(* IEC 61131-3 sources: SmartHomeNew/ (part 2) *)

(* ---- GVL_DEBUG_VIEW.gvl ---- *)
VAR_GLOBAL
    D_Current_Time_MS : UDINT := 0;

    D_Safety_Mode : E_Safety_Mode := NORMAL;
    D_Safety_Active : BOOL := FALSE;
    D_Recovery_Phase : E_Recovery_Phase := IDLE;
    D_Recovery_Active : BOOL := FALSE;
    D_Recovery_Exit_Allowed : BOOL := FALSE;
    D_Authority_Revocation_Active : BOOL := FALSE;
    D_Authority_Restoration_Allowed : BOOL := FALSE;
    D_Authority_Restoration_Completed : BOOL := FALSE;

    D_Current_Scenario : STRING(255) := '';
    D_Behavior_Reason : STRING(255) := '';
    D_Score_Night : INT := 0;
    D_Score_Preheat : INT := 0;
    D_Score_VentBoost : INT := 0;
    D_Score_AccessSecure : INT := 0;
    D_Intent_Night : BOOL := FALSE;
    D_Intent_Comfort : BOOL := FALSE;
    D_Intent_VentBoost : BOOL := FALSE;
    D_Intent_AccessSecure : BOOL := FALSE;

    D_Heating_Block : BOOL := FALSE;
    D_Vent_Stop : BOOL := FALSE;
    D_Water_Block : BOOL := FALSE;
    D_Access_Open_Active : BOOL := FALSE;

    D_Global_Reason : STRING(255) := '';
    D_Behavior_Why_Active : STRING(255) := '';
    D_Heating_Why_Blocked : STRING(255) := '';
    D_Vent_Why_Stopped : STRING(255) := '';
    D_Water_Why_Closed : STRING(255) := '';
    D_Access_Why_Opened : STRING(255) := '';

    D_Main_VentBoost_Zone : INT := 0;
    D_Main_VentBoost_Zone_Weight : REAL := 0.0;
    D_Main_VentBoost_Zone_Confidence : REAL := 0.0;
    D_Max_VentBoost_Zone_Weight : REAL := 0.0;
    D_Min_VentBoost_Zone_Weight : REAL := 0.0;

    // MAIN phase feedback summary.
    D_Main_Phase_Current : UINT := 0;
    D_Main_Phase_Critical_Executed : BOOL := FALSE;
    D_Main_Phase_Critical_Valid : BOOL := FALSE;
    D_Main_Phase_Observability_Executed : BOOL := FALSE;
    D_Main_Phase_Observability_Valid : BOOL := FALSE;
    D_Main_Phase_Any_Invalid : BOOL := FALSE;
    D_Main_Phase_Any_Skipped_By_Design : BOOL := FALSE;
    D_Main_Phase_Status_Code : UINT := 0;
    D_Main_Phase_Status_Text : STRING(160) := '';

    // Domain execution policy summary.
    D_Domain_Policy_Any_Critical : BOOL := FALSE;
    D_Domain_Policy_Any_Periodic : BOOL := FALSE;
    D_Domain_Policy_Any_Periodic_Due : BOOL := FALSE;
    D_Domain_Policy_Any_Idle : BOOL := FALSE;
    D_Domain_Policy_Status_Code : UINT := 0;
    D_Domain_Policy_Status_Text : STRING(160) := '';

    D_Access_Mode : UINT := 0;
    D_Access_Critical_Run : BOOL := FALSE;
    D_Access_Periodic_Run : BOOL := FALSE;
    D_Access_Periodic_Due : BOOL := FALSE;
    D_Access_Idle_By_Design : BOOL := FALSE;

    D_Lighting_Mode : UINT := 0;
    D_Lighting_Critical_Run : BOOL := FALSE;
    D_Lighting_Periodic_Run : BOOL := FALSE;
    D_Lighting_Periodic_Due : BOOL := FALSE;
    D_Lighting_Idle_By_Design : BOOL := FALSE;

    D_Water_Mode : UINT := 0;
    D_Water_Critical_Run : BOOL := FALSE;
    D_Water_Periodic_Run : BOOL := FALSE;
    D_Water_Periodic_Due : BOOL := FALSE;
    D_Water_Idle_By_Design : BOOL := FALSE;

    D_Heating_Mode : UINT := 0;
    D_Heating_Critical_Run : BOOL := FALSE;
    D_Heating_Periodic_Run : BOOL := FALSE;
    D_Heating_Periodic_Due : BOOL := FALSE;
    D_Heating_Idle_By_Design : BOOL := FALSE;

    D_Vent_Mode : UINT := 0;
    D_Vent_Critical_Run : BOOL := FALSE;
    D_Vent_Periodic_Run : BOOL := FALSE;
    D_Vent_Periodic_Due : BOOL := FALSE;
    D_Vent_Idle_By_Design : BOOL := FALSE;

    D_Simulation_Mode : UINT := 0;
    D_Simulation_Run_Allowed : BOOL := FALSE;
    D_Simulation_Periodic_Due : BOOL := FALSE;
    D_Simulation_Idle_By_Design : BOOL := FALSE;

    // Domain execution validation summary.
    D_Domain_Validation_Executed : BOOL := FALSE;
    D_Domain_Validation_Valid : BOOL := FALSE;
    D_Domain_Validation_Any_Stale_Output_Risk : BOOL := FALSE;
    D_Domain_Validation_Any_Policy_Mismatch : BOOL := FALSE;
    D_Access_Stale_Output_Risk : BOOL := FALSE;
    D_Lighting_Stale_Output_Risk : BOOL := FALSE;
    D_Water_Stale_Output_Risk : BOOL := FALSE;
    D_Heating_Stale_Output_Risk : BOOL := FALSE;
    D_Vent_Stale_Output_Risk : BOOL := FALSE;
    D_Domain_Validation_Status_Code : UINT := 0;
    D_Domain_Validation_Status_Text : STRING(160) := '';

    // Runtime scenario validation summary.
    D_Runtime_Scenario_Validation_Executed : BOOL := FALSE;
    D_Runtime_Scenario_Validation_Valid : BOOL := FALSE;
    D_Runtime_Scenario_Any_Context_Invalid : BOOL := FALSE;
    D_Runtime_Idle_Context_Active : BOOL := FALSE;
    D_Runtime_Security_Context_Active : BOOL := FALSE;
    D_Runtime_Away_Context_Active : BOOL := FALSE;
    D_Runtime_Presence_Context_Active : BOOL := FALSE;
    D_Runtime_Fire_Context_Active : BOOL := FALSE;
    D_Runtime_Gas_Context_Active : BOOL := FALSE;
    D_Runtime_Leak_Context_Active : BOOL := FALSE;
    D_Runtime_Global_Stop_Context_Active : BOOL := FALSE;
    D_Runtime_Freeze_Context_Active : BOOL := FALSE;
    D_Runtime_Heating_Context_Valid : BOOL := FALSE;
    D_Runtime_Vent_Context_Valid : BOOL := FALSE;
    D_Runtime_Access_Context_Valid : BOOL := FALSE;
    D_Runtime_Global_Stop_Context_Valid : BOOL := FALSE;
    D_Runtime_Scenario_Status_Code : UINT := 0;
    D_Runtime_Scenario_Status_Text : STRING(160) := '';

    // Runtime physical IO validation summary.
    D_Runtime_IO_Validation_Executed : BOOL := FALSE;
    D_Runtime_IO_Validation_Valid : BOOL := FALSE;
    D_Runtime_IO_Any_Invalid : BOOL := FALSE;
    D_Runtime_IO_Fire_Valid : BOOL := FALSE;
    D_Runtime_IO_Gas_Valid : BOOL := FALSE;
    D_Runtime_IO_Leak_Valid : BOOL := FALSE;
    D_Runtime_IO_Global_Stop_Valid : BOOL := FALSE;
    D_Runtime_IO_Inactive_PLC_Valid : BOOL := FALSE;
    D_Runtime_IO_Freeze_Valid : BOOL := FALSE;
    D_Runtime_IO_Status_Code : UINT := 0;
    D_Runtime_IO_Status_Text : STRING(160) := '';

    // HMI / dashboard sensor quality view.
    D_Input_Source_Valid : BOOL := FALSE;
    D_Input_Degraded : BOOL := FALSE;
    D_Sensor_Fault : BOOL := FALSE;
    D_Validation_Failed : BOOL := FALSE;
    D_Anomaly_Detected : BOOL := FALSE;
    D_Validation_Reason : STRING(120) := '';
    D_Anomaly_Reason : STRING(120) := '';
    D_Last_Invalid_Zone : INT := 0;
    D_Min_Zone_Confidence : REAL := 1.0;
    D_Worst_Zone : INT := 0;

    // Runtime diagnostics formerly stored in legacy GVL_TEST.
    D_Ownership_Violation : BOOL := FALSE;

    D_Adapt_Profile : E_Adapt_Profile := ADAPT_PROFILE_BALANCED;
    D_Adapt_Profile_Text : STRING(32) := 'BALANCED';

    D_Last_Trace_Text : STRING(120) := '';
    D_Last_Trace_Time_MS : UDINT := 0;
    D_Last_Trace_Reason : E_System_Reason_Code := REASON_NONE;
END_VAR

(* ---- GVL_DIAGNOSTICS_EXT.gvl ---- *)
{attribute 'qualified_only'}
VAR_GLOBAL
    // Health scores (0..1)
    G_Health_Heating : REAL := 1.0;
    G_Health_Safety : REAL := 1.0;
    G_Health_IO : REAL := 1.0;

    // Error counters
    G_Error_Count_Heating : UDINT := 0;
    G_Error_Count_Safety : UDINT := 0;
    G_Error_Count_IO : UDINT := 0;

    // Last error timestamps
    G_Last_Error_Time_Heating : UDINT := 0;
    G_Last_Error_Time_Safety : UDINT := 0;
    G_Last_Error_Time_IO : UDINT := 0;

    // Timing
    G_Last_Update_Time : UDINT := 0;

    // Cycle / watchdog statistics (interval between diagnostics executions)
    G_Cycle_Expected_MS : UDINT := 250;
    G_Cycle_Warning_MS : UDINT := 375;
    G_Cycle_Critical_MS : UDINT := 500;
    G_Cycle_Last_MS : UDINT := 0;
    G_Cycle_Max_MS : UDINT := 0;
    G_Cycle_Min_MS : UDINT := 0;
    G_Cycle_Avg_MS : REAL := 0.0;
    G_Cycle_Sample_Count : UDINT := 0;
    G_Cycle_Overrun_Count : UDINT := 0;
    G_Cycle_Critical_Count : UDINT := 0;
    G_Cycle_Last_Overrun_MS : UDINT := 0;
    G_Cycle_Last_Overrun_Time_MS : UDINT := 0;
    G_Cycle_Overrun_Active : BOOL := FALSE;
    G_Cycle_Critical_Active : BOOL := FALSE;

    // Compact degraded state mirrors.
    G_Heating_State : INT := 0; // 0=OK,1=DEGRADED,2=CRITICAL
    G_Safety_State : INT := 0;
    G_IO_State : INT := 0;
END_VAR

(* ---- GVL_Distributed_Authority.gvl ---- *)
{attribute 'qualified_only'}
VAR_GLOBAL RETAIN
    G_Authority_State : ST_Distributed_Authority_State;

    G_Master_Controller_Id : UINT;
    G_Backup_Controller_Id : UINT;

    G_Authority_Lease_Start_MS : UDINT;
    G_Authority_Lease_Duration_MS : UDINT := 30000;
END_VAR

VAR_GLOBAL
    G_Runtime_Valid : BOOL;
    G_Last_Update_MS : UDINT;

    G_Split_Brain_Blocked : BOOL;
    G_Distributed_Safety_Barrier_OK : BOOL;

    G_Status_Code : UINT;
    G_Status_Text : STRING(160);
END_VAR

(* ---- GVL_DISTRIBUTED_COMMIT.gvl ---- *)
VAR_GLOBAL
    // ======================================================
    // DISTRIBUTED PUBLICATION COMMIT STATE
    // ======================================================
    // Deterministic peer publication commit handshake foundation.
    // Publication-continuity governance only.
    // Does not invalidate runtime barrier, PLC fencing
    // or local immutable snapshot authority.
    // ======================================================

    Distributed_Commit_Epoch : ULINT := 0;
    Distributed_Commit_Reconciliation_Epoch : ULINT := 0;

    Local_Publication_Commit_Epoch : ULINT := 0;
    Peer_Publication_Commit_Epoch : ULINT := 0;

    Local_Prepare_Epoch : ULINT := 0;
    Peer_Prepare_Epoch : ULINT := 0;

    Local_Commit_Token : ULINT := 0;
    Peer_Commit_Token : ULINT := 0;

    Publication_Prepare_Active : BOOL := FALSE;
    Publication_Prepare_Valid : BOOL := FALSE;
    Publication_Commit_Requested : BOOL := FALSE;
    Publication_Commit_Confirmed : BOOL := FALSE;

    Peer_Commit_Ack_Valid : BOOL := FALSE;
    Peer_Commit_Ack_Expired : BOOL := FALSE;
    Peer_Commit_Mismatch : BOOL := FALSE;
    Peer_Commit_Replay_Detected : BOOL := FALSE;
    Peer_Commit_Missing : BOOL := FALSE;

    Commit_Lease_Active : BOOL := FALSE;
    Commit_Lease_Expired : BOOL := FALSE;
    Commit_Timeout_MS : UDINT := 5000;

    Local_Commit_Last_Refresh_MS : UDINT := 0;
    Peer_Commit_Last_Refresh_MS : UDINT := 0;
    Commit_Last_Reconciliation_MS : UDINT := 0;

    Distributed_Commit_Valid : BOOL := FALSE;
    Distributed_Commit_Quarantine_Active : BOOL := FALSE;

    Distributed_Commit_Last_Error_Code : UDINT := 0;
    Distributed_Commit_Last_Error_Text : STRING(160) := '';
END_VAR

(* ---- GVL_DISTRIBUTED_EPOCH.gvl ---- *)
VAR_GLOBAL
    // ======================================================
    // DISTRIBUTED EPOCH CONSISTENCY STATE
    // ======================================================
    // Centralized peer epoch reconciliation foundation.
    // Prevents distributed stale authority and split-brain continuity.
    // ======================================================

    Distributed_Epoch : ULINT := 0;
    Distributed_Reconciliation_Epoch : ULINT := 0;

    Local_Runtime_Epoch : ULINT := 0;
    Peer_Runtime_Epoch : ULINT := 0;

    Local_Snapshot_Epoch : ULINT := 0;
    Peer_Snapshot_Epoch : ULINT := 0;

    Local_Boot_Generation : ULINT := 0;
    Peer_Boot_Generation : ULINT := 0;

    Local_Fencing_Token : ULINT := 0;
    Peer_Fencing_Token : ULINT := 0;

    Distributed_Epoch_Consistent : BOOL := FALSE;
    Distributed_Reconciliation_Valid : BOOL := FALSE;
    Distributed_Publication_Allowed : BOOL := FALSE;

    Peer_Lease_Active : BOOL := FALSE;
    Peer_Lease_Expired : BOOL := FALSE;
    Peer_Lease_Timeout_MS : UDINT := 5000;

    Peer_Last_Refresh_MS : UDINT := 0;
    Peer_Last_Reconciliation_MS : UDINT := 0;

    Peer_Snapshot_Stale : BOOL := FALSE;
    Peer_Runtime_Stale : BOOL := FALSE;
    Peer_Boot_Mismatch : BOOL := FALSE;
    Peer_Fencing_Conflict : BOOL := FALSE;
    Peer_Semantic_Continuity_Lost : BOOL := FALSE;

    Distributed_Quarantine_Active : BOOL := FALSE;

    Distributed_Last_Error_Code : UDINT := 0;
    Distributed_Last_Error_Text : STRING(160) := '';
END_VAR

(* ---- GVL_Distributed_Orchestration.gvl ---- *)
{attribute 'qualified_only'}
VAR_GLOBAL
    G_Topology_Domain : ARRAY[1..32] OF ST_Distributed_Topology_Domain;
    G_Orchestration_State : ST_Distributed_Orchestration_State;
END_VAR

VAR_GLOBAL RETAIN
    G_Last_Distributed_Sequence_Id : UDINT;
END_VAR

VAR_GLOBAL
    G_Runtime_Valid : BOOL;
    G_Last_Update_MS : UDINT;

    G_Cross_Node_Isolation_Active : BOOL;
    G_Cross_Node_Recovery_Active : BOOL;
    G_Cross_Node_Rollback_Active : BOOL;

    G_Distributed_Projection_Healthy : BOOL;
    G_Distributed_Scheduler_Healthy : BOOL;

    G_Status_Code : UINT;
    G_Status_Text : STRING(160);
END_VAR

(* ---- GVL_Distributed_Projection_Ownership.gvl ---- *)
{attribute 'qualified_only'}
VAR_GLOBAL RETAIN
    G_Projection_Ownership : ARRAY[1..128] OF ST_Distributed_Projection_Ownership;
END_VAR

VAR_GLOBAL
    G_Runtime_Valid : BOOL;
    G_Last_Update_MS : UDINT;

    G_Any_Ownership_Conflict : BOOL;
    G_Any_Ownership_Stale : BOOL;
    G_Any_Projection_Blocked : BOOL;

    G_Status_Code : UINT;
    G_Status_Text : STRING(160);
END_VAR

(* ---- GVL_Distributed_Runtime.gvl ---- *)
{attribute 'qualified_only'}
VAR_GLOBAL RETAIN
    // Keep only compact continuity metadata in non-volatile memory.
    // Runtime node/session/message state is rebuilt by the distributed
    // supervisor chain during cyclic execution and must not consume RETAIN.
    G_Last_Replication_Sequence_Id : UDINT;
END_VAR

VAR_GLOBAL
    G_Local_Node_State : ST_Distributed_Runtime_Node_State;
    G_Remote_Node_State : ARRAY[1..8] OF ST_Distributed_Runtime_Node_State;

    G_Replication_TX : ARRAY[1..64] OF ST_Distributed_Runtime_Message;
    G_Replication_RX : ARRAY[1..64] OF ST_Distributed_Runtime_Message;

    G_Runtime_Valid : BOOL;
    G_Last_Update_MS : UDINT;

    G_Any_Remote_Node_Degraded : BOOL;
    G_Any_Remote_Node_Offline : BOOL;
    G_Split_Brain_Suspected : BOOL;

    G_Distributed_Authority_Healthy : BOOL;
    G_Distributed_Replication_Healthy : BOOL;

    G_Status_Code : UINT;
    G_Status_Text : STRING(160);
END_VAR

(* ---- GVL_DISTRIBUTED_SNAPSHOT.gvl ---- *)
VAR_GLOBAL
    // ======================================================
    // DISTRIBUTED IMMUTABLE SNAPSHOT STATE
    // ======================================================
    // Peer immutable publication snapshot reconciliation.
    // Publication-authoritative only: does not invalidate
    // runtime barrier, PLC fencing or local snapshot freeze.
    // ======================================================

    Distributed_Snapshot_Epoch : ULINT := 0;
    Distributed_Snapshot_Reconciliation_Epoch : ULINT := 0;

    Local_Distributed_Snapshot_Epoch : ULINT := 0;
    Peer_Distributed_Snapshot_Epoch : ULINT := 0;

    Local_Runtime_Snapshot_Epoch : ULINT := 0;
    Peer_Runtime_Snapshot_Epoch : ULINT := 0;

    Local_Publication_Epoch : ULINT := 0;
    Peer_Publication_Epoch : ULINT := 0;

    Distributed_Snapshot_Frozen : BOOL := FALSE;
    Peer_Snapshot_Immutable : BOOL := FALSE;

    Distributed_Publication_Reconciled : BOOL := FALSE;
    Distributed_Publication_Freeze_Valid : BOOL := FALSE;
    Distributed_Snapshot_Consistent : BOOL := FALSE;

    Peer_Publication_Stale : BOOL := FALSE;
    Peer_Snapshot_Not_Immutable : BOOL := FALSE;
    Peer_Publication_Divergence : BOOL := FALSE;
    Peer_Publication_Reconciliation_Lost : BOOL := FALSE;

    Distributed_Snapshot_Quarantine_Active : BOOL := FALSE;

    Peer_Snapshot_Last_Refresh_MS : UDINT := 0;
    Peer_Snapshot_Lease_Active : BOOL := FALSE;
    Peer_Snapshot_Lease_Expired : BOOL := FALSE;
    Peer_Snapshot_Lease_Timeout_MS : UDINT := 5000;

    Distributed_Snapshot_Last_Error_Code : UDINT := 0;
    Distributed_Snapshot_Last_Error_Text : STRING(160) := '';
END_VAR

(* ---- GVL_DOMAIN_EXECUTION_POLICY.gvl ---- *)
{attribute 'qualified_only'}
VAR_GLOBAL
    // Domain execution policy. Observational first layer.
    // This GVL classifies when a domain needs critical, periodic or idle execution.
    // It does not directly control physical outputs.

    G_Last_Update_MS : UDINT := 0;

    // Scenario/context classification.
    G_Security_Context_Active : BOOL := FALSE;
    G_Away_Context_Active : BOOL := FALSE;
    G_Presence_Context_Active : BOOL := FALSE;
    G_Emergency_Context_Active : BOOL := FALSE;

    // Periodic observation intervals.
    Access_Periodic_Interval_MS : UDINT := 1000;
    Lighting_Periodic_Interval_MS : UDINT := 1000;
    Water_Periodic_Interval_MS : UDINT := 1000;
    Heating_Periodic_Interval_MS : UDINT := 5000;
    Vent_Periodic_Interval_MS : UDINT := 3000;
    Simulation_Periodic_Interval_MS : UDINT := 1000;

    // Access.
    Access_Critical_Run : BOOL := FALSE;
    Access_Periodic_Run : BOOL := FALSE;
    Access_Periodic_Due : BOOL := FALSE;
    Access_Idle_By_Design : BOOL := FALSE;

    // Lighting.
    Lighting_Critical_Run : BOOL := FALSE;
    Lighting_Periodic_Run : BOOL := FALSE;
    Lighting_Periodic_Due : BOOL := FALSE;
    Lighting_Idle_By_Design : BOOL := FALSE;

    // Water.
    Water_Critical_Run : BOOL := FALSE;
    Water_Periodic_Run : BOOL := FALSE;
    Water_Periodic_Due : BOOL := FALSE;
    Water_Idle_By_Design : BOOL := FALSE;

    // Heating.
    Heating_Critical_Run : BOOL := FALSE;
    Heating_Periodic_Run : BOOL := FALSE;
    Heating_Periodic_Due : BOOL := FALSE;
    Heating_Idle_By_Design : BOOL := FALSE;

    // Ventilation.
    Vent_Critical_Run : BOOL := FALSE;
    Vent_Periodic_Run : BOOL := FALSE;
    Vent_Periodic_Due : BOOL := FALSE;
    Vent_Idle_By_Design : BOOL := FALSE;

    // Simulation.
    Simulation_Context_Active : BOOL := FALSE;
    Simulation_Run_Allowed : BOOL := FALSE;
    Simulation_Periodic_Due : BOOL := FALSE;
    Simulation_Idle_By_Design : BOOL := FALSE;

    // Summary.
    Any_Critical_Run : BOOL := FALSE;
    Any_Periodic_Run : BOOL := FALSE;
    Any_Periodic_Due : BOOL := FALSE;
    Any_Idle_By_Design : BOOL := FALSE;
    Status_Code : UINT := 0;
    Status_Text : STRING(160) := '';
END_VAR

(* ---- GVL_DOMAIN_EXECUTION_VALIDATION.gvl ---- *)
{attribute 'qualified_only'}
VAR_GLOBAL
    // Domain execution validation. Observational only.
    // Detects policy/output mismatches before runtime gating is trusted.

    G_Last_Update_MS : UDINT := 0;
    G_Validation_Executed : BOOL := FALSE;
    G_Validation_Valid : BOOL := TRUE;

    Access_Stale_Output_Risk : BOOL := FALSE;
    Lighting_Stale_Output_Risk : BOOL := FALSE;
    Water_Stale_Output_Risk : BOOL := FALSE;
    Heating_Stale_Output_Risk : BOOL := FALSE;
    Vent_Stale_Output_Risk : BOOL := FALSE;

    Any_Stale_Output_Risk : BOOL := FALSE;
    Any_Policy_Mismatch : BOOL := FALSE;
    Status_Code : UINT := 0;
    Status_Text : STRING(160) := '';
END_VAR

(* ---- GVL_ENERGY_ISOLATION_CAUSALITY_FABRIC.gvl ---- *)
VAR_GLOBAL
    Energy_Isolation_Causality_Valid : BOOL := FALSE;
    Energy_Isolation_Causality_Granted : BOOL := FALSE;

    Physical_Energy_Isolation_Valid : BOOL := FALSE;
    Unsafe_Energy_Propagation_Prevented : BOOL := FALSE;
    CrossDomain_Power_Segmentation_Canonical : BOOL := FALSE;
    Energy_Isolation_Lineage_Coherent : BOOL := FALSE;

    Energy_Causality_Grounded : BOOL := FALSE;
    Distributed_Energy_Isolation_Consensus : BOOL := FALSE;

    Residual_Energy_Leakage_Detected : BOOL := FALSE;
    CrossDomain_Power_Backfeed_Detected : BOOL := FALSE;
    SplitEnergy_Topology_Detected : BOOL := FALSE;
    Unsafe_Energy_Propagation_Detected : BOOL := FALSE;

    Energy_Isolation_Epoch : UDINT := 0;
END_VAR

(* ---- GVL_EPISTEMIC_INTEGRITY_FABRIC.gvl ---- *)
VAR_GLOBAL
    // Global deterministic epistemic integrity authority.
    Epistemic_Integrity_Valid : BOOL := FALSE;
    Epistemic_Integrity_Granted : BOOL := FALSE;
    Epistemic_Integrity_Quarantine_Active : BOOL := TRUE;

    // Physical reality anchoring proofs.
    Physical_Reality_Model_Coherent : BOOL := FALSE;
    Sensor_Truth_Consensus_Valid : BOOL := FALSE;
    Telemetry_Reality_Alignment_Stable : BOOL := FALSE;
    Distributed_Reality_Model_Consistent : BOOL := FALSE;
    Causal_Model_Physically_Valid : BOOL := FALSE;

    // Long-term epistemic integrity.
    Historical_Reality_Anchoring_Valid : BOOL := FALSE;
    Physical_Truth_Lineage_Coherent : BOOL := FALSE;
    Reality_Model_Drift_Bounded : BOOL := FALSE;
    Semantic_To_Physical_Causality_Valid : BOOL := FALSE;

    // Epistemic split-brain detectors.
    Physically_False_Consensus_Detected : BOOL := FALSE;
    Telemetry_Corruption_Coherent_Detected : BOOL := FALSE;
    Historical_Reality_Divergence_Detected : BOOL := FALSE;
    Sensor_Trust_Erosion_Detected : BOOL := FALSE;
    Causal_Model_Poisoning_Detected : BOOL := FALSE;
    LongTerm_Epistemic_Drift_Detected : BOOL := FALSE;

    // Epistemic epochs.
    Epistemic_Integrity_Epoch : UDINT := 0;
    Epistemic_Integrity_Epoch_Coherent : BOOL := FALSE;

    // Temporal authority.
    Epistemic_Integrity_Last_Update_MS : UDINT := 0;
    Epistemic_Integrity_Lease_Expired : BOOL := TRUE;

    // Diagnostics.
    Epistemic_Integrity_Last_Error_Code : UDINT := 0;
    Epistemic_Integrity_Last_Error_Text : STRING(160) := '';
    Epistemic_Integrity_Invalidation_Count : UDINT := 0;
END_VAR

(* ---- GVL_EXECUTION_PROGRESS_CAUSALITY_FABRIC.gvl ---- *)
VAR_GLOBAL
    Execution_Progress_Causality_Valid : BOOL := FALSE;
    Execution_Progress_Causality_Granted : BOOL := FALSE;

    Progress_Causality_Grounded : BOOL := FALSE;
    Deterministic_Execution_Continuation_Valid : BOOL := FALSE;
    Progress_Lineage_Coherent : BOOL := FALSE;

    Distributed_Progress_Convergence_Valid : BOOL := FALSE;
    Progress_Timeline_Monotonic : BOOL := FALSE;

    Distributed_Execution_Stall_Detected : BOOL := FALSE;
    Execution_Progress_Divergence_Detected : BOOL := FALSE;
    Recovery_Progress_Oscillation_Detected : BOOL := FALSE;

    Execution_Progress_Epoch : UDINT := 0;
END_VAR

(* ---- GVL_EXECUTION_PROJECTION_INTEGRITY_FABRIC.gvl ---- *)
VAR_GLOBAL
    // Deterministic execution projection integrity governance.
    Execution_Projection_Integrity_Valid : BOOL := FALSE;
    Execution_Projection_Integrity_Granted : BOOL := FALSE;
    Execution_Projection_Integrity_Quarantine_Active : BOOL := TRUE;

    // Governance-to-execution projection proofs.
    Execution_Authority_Projection_Consistent : BOOL := FALSE;
    CrossDomain_Actuation_Enforcement_Aligned : BOOL := FALSE;
    Physical_Execution_Governance_Canonical : BOOL := FALSE;
    Actuation_Surface_Consensus_Valid : BOOL := FALSE;
    Execution_Projection_Lineage_Coherent : BOOL := FALSE;

    // Execution enforcement integrity.
    Runtime_Actuation_Projection_Stable : BOOL := FALSE;
    Distributed_Execution_Equivalence_Valid : BOOL := FALSE;
    Execution_Governance_Causality_Grounded : BOOL := FALSE;
    Physical_Enforcement_Timeline_Monotonic : BOOL := FALSE;

    // Execution projection split-brain detectors.
    Execution_Projection_Divergence_Detected : BOOL := FALSE;
    Actuation_Path_Authority_Bypass_Detected : BOOL := FALSE;
    CrossDomain_Enforcement_Fork_Detected : BOOL := FALSE;
    Canonical_Governance_Execution_Lost : BOOL := FALSE;
    Runtime_Execution_Lineage_Drift_Detected : BOOL := FALSE;
    Distributed_Actuation_Reality_Fork_Detected : BOOL := FALSE;

    // Execution epochs.
    Execution_Projection_Integrity_Epoch : UDINT := 0;
    Execution_Projection_Integrity_Epoch_Coherent : BOOL := FALSE;

    // Temporal authority.
    Execution_Projection_Integrity_Last_Update_MS : UDINT := 0;
    Execution_Projection_Integrity_Lease_Expired : BOOL := TRUE;

    // Diagnostics.
    Execution_Projection_Integrity_Last_Error_Code : UDINT := 0;
    Execution_Projection_Integrity_Last_Error_Text : STRING(160) := '';
    Execution_Projection_Integrity_Invalidation_Count : UDINT := 0;
END_VAR

(* ---- GVL_External_Monitoring.gvl ---- *)
VAR_GLOBAL
    // === EXTERNAL SHADOW POLICY CONTRACT ===
    G_Shadow_Any_Alert_Active : BOOL;
    G_Shadow_CO_Active : BOOL;
    G_Shadow_Methane_Active : BOOL;
    G_Shadow_Smoke_Active : BOOL;

    G_Shadow_CO_Healthy : BOOL;
    G_Shadow_Methane_Healthy : BOOL;
    G_Shadow_Smoke_Healthy : BOOL;

    G_Shadow_Dominant_Channel : STRING(32);
    G_Shadow_Policy_Summary_Text : STRING(160);
    G_Shadow_Recent_Activity_Text : STRING(160);
    G_Shadow_Rate_Summary_Text : STRING(160);
    G_Shadow_Rate_Alert_Text : STRING(160);

    G_Shadow_Total_Fallback_Count : UDINT;
    G_Shadow_Total_Recovery_Count : UDINT;

    G_Shadow_Rate_Fallback_Per_Hour : REAL;
    G_Shadow_Rate_Recovery_Per_Hour : REAL;

    G_Shadow_Rate_Alert_Active : BOOL;
END_VAR

(* ---- GVL_FILE_ARCHIVE.gvl ---- *)
{attribute 'qualified_only'}
VAR_GLOBAL
    // Runtime interface for future file/CSV archive integration.
    // No direct file/USB write is implemented here. Concrete CODESYS file
    // libraries, USB/flash paths, CSV formatting and buffering are connected
    // during the porting/module-selection stage.

    G_Archive_Interface_Enabled : BOOL := FALSE;
    G_File_Archive_Target_Code : BYTE := 0; // 0=none, 1=PLC file/flash, 2=USB, 3=gateway
    G_USB_Target_Available : BOOL := FALSE;
    G_PLC_File_Target_Available : BOOL := FALSE;
    G_Gateway_Target_Available : BOOL := FALSE;

    G_CSV_Write_Enabled : BOOL := FALSE;
    G_Write_Event_CSV_Request : BOOL := FALSE;
    G_Write_Trend_CSV_Request : BOOL := FALSE;
    G_Write_BlackBox_CSV_Request : BOOL := FALSE;
    G_Write_Config_Backup_Request : BOOL := FALSE;

    // Automatic configuration backup scheduler.
    // Default trigger is 03:00 local/effective time. The scheduler publishes
    // the same one-shot config backup request as HMI/gateway paths.
    G_Auto_Config_Backup_Enabled : BOOL := FALSE;
    G_Auto_Config_Backup_Time_Of_Day_MS : UDINT := 10800000;
    G_Auto_Config_Backup_Last_Day_Of_Week : INT := 0;
    G_Auto_Config_Backup_Last_Request_MS : UDINT := 0;
    G_Auto_Config_Backup_Last_Status_Text : STRING(200) := '';

    G_Write_Busy : BOOL := FALSE;
    G_Write_Done : BOOL := FALSE;
    G_Write_Error : BOOL := FALSE;
    G_Last_Error_Code : UDINT := 0;
    G_Last_Status_Text : STRING(200) := '';
    G_Last_Write_MS : UDINT := 0;
END_VAR

(* ---- GVL_FILE_ARCHIVE_HMI.gvl ---- *)
{attribute 'qualified_only'}
VAR_GLOBAL
    // HMI intent surface for file/archive operations.
    // This is a request/configuration surface only. The actual runtime status is
    // published by GVL_FILE_ARCHIVE and mirrored to GVL_HMI by PRG_HMI_Dashboard.

    // Archive configuration request.
    G_Set_Archive_Config_Req : BOOL := FALSE;
    G_Archive_Interface_Enabled : BOOL := FALSE;
    G_CSV_Write_Enabled : BOOL := FALSE;
    G_File_Archive_Target_Code : BYTE := 0; // 0=none, 1=PLC file/flash, 2=USB, 3=gateway

    // Automatic configuration backup schedule request.
    // Time is milliseconds from start of effective day, default 03h00.
    G_Set_Auto_Config_Backup_Req : BOOL := FALSE;
    G_Auto_Config_Backup_Enabled : BOOL := FALSE;
    G_Auto_Config_Backup_Time_Of_Day_MS : UDINT := 10800000;

    // One-shot archive write requests.
    G_Write_Event_CSV_Req : BOOL := FALSE;
    G_Write_Trend_CSV_Req : BOOL := FALSE;
    G_Write_BlackBox_CSV_Req : BOOL := FALSE;
    G_Write_Config_Backup_Req : BOOL := FALSE;

    // Applicator feedback.
    G_Last_Status_Text : STRING(200) := '';
    G_Last_Error : BOOL := FALSE;
    G_Last_Error_Code : UDINT := 0;
    G_Last_Update_MS : UDINT := 0;
END_VAR

(* ---- GVL_Forensic_Journal.gvl ---- *)
{attribute 'qualified_only'}
VAR_GLOBAL
    G_Journal : ARRAY[1..256] OF ST_Forensic_Journal_Record;
END_VAR

VAR_GLOBAL RETAIN
    G_Write_Index : UINT;
    G_Last_Event_Id : UDINT;
END_VAR

VAR_GLOBAL
    G_Runtime_Valid : BOOL;
    G_Last_Update_MS : UDINT;

    G_Last_Activation_Event_Id : UDINT;
    G_Last_Rollback_Event_Id : UDINT;
    G_Last_Recovery_Event_Id : UDINT;
    G_Last_Restart_Event_Id : UDINT;

    G_Status_Code : UINT;
    G_Status_Text : STRING(160);
END_VAR

(* ---- GVL_GATEWAY.gvl ---- *)
{attribute 'qualified_only'}
VAR_GLOBAL
    G_Gateway_Command : ST_Gateway_Command;
    G_Gateway_Command_Received : BOOL;
    G_Gateway_Telegram_Msg : STRING(200);
    G_Gateway_Send_Telegram : BOOL;
    G_Gateway_HMI_Status_Message : STRING(200);
    G_Gateway_Ping_OK : BOOL;
    G_Gateway_Data_Ready : BOOL;
    G_Gateway_Modbus_Registers : ARRAY[0..GVL_CONSTANTS.C_MAX_MODBUS_REGISTERS-1] OF WORD;
END_VAR

(* ---- GVL_GLOBAL_AUTHORITY_SYNC.gvl ---- *)
VAR_GLOBAL
    // Global synchronized authority fabric.
    Global_Authority_Sync_Valid : BOOL := FALSE;
    Global_Authority_Sync_Granted : BOOL := FALSE;
    Global_Authority_Sync_Quarantine_Active : BOOL := TRUE;

    // Cross-domain authority coherence.
    Heating_Authority_Coherent : BOOL := FALSE;
    Ventilation_Authority_Coherent : BOOL := FALSE;
    Water_Authority_Coherent : BOOL := FALSE;
    Access_Authority_Coherent : BOOL := FALSE;
    Lighting_Authority_Coherent : BOOL := FALSE;

    // Global causality synchronization.
    Cross_Domain_Epoch_Coherent : BOOL := FALSE;
    Distributed_Authority_Generation_Coherent : BOOL := FALSE;
    Global_Causality_Timeline_Stable : BOOL := FALSE;
    Multi_Domain_Recovery_Coherent : BOOL := FALSE;

    // Cross-domain split-brain detection.
    Authority_Epoch_Fragmentation_Detected : BOOL := FALSE;
    Partial_Recovery_SplitBrain_Detected : BOOL := FALSE;
    Cross_Domain_Replay_Skew_Detected : BOOL := FALSE;
    Distributed_Authority_Divergence_Detected : BOOL := FALSE;
    Global_Causality_Desynchronization_Detected : BOOL := FALSE;
    Multi_Domain_Chronology_Drift_Detected : BOOL := FALSE;

    // Synchronized authority epochs.
    Global_Authority_Epoch : UDINT := 0;
    Global_Authority_Epoch_Coherent : BOOL := FALSE;

    // Temporal synchronization authority.
    Global_Authority_Last_Update_MS : UDINT := 0;
    Global_Authority_Lease_Expired : BOOL := TRUE;

    // Diagnostics.
    Global_Authority_Last_Error_Code : UDINT := 0;
    Global_Authority_Last_Error_Text : STRING(160) := '';
    Global_Authority_Invalidation_Count : UDINT := 0;
END_VAR

(* ---- GVL_HA_SESSION_REPLICATION.gvl ---- *)
VAR_GLOBAL
    // ======================================================
    // HA SESSION REPLICATION BOUNDARY
    // ======================================================
    // Dedicated high-availability session replication boundary.
    //
    // Purpose:
    // isolate peer-session replication from:
    // - Modbus transport runtime
    // - IO runtime
    // - distributed reconciliation governors
    //
    // Ownership:
    // - PRG_Peer_Session_Publication exports canonical local state
    // - HA/session transport publishes replicated remote state
    // - PRG_Distributed_Peer_Ingestion consumes replicated state
    // - PRG_Distributed_Snapshot_Ingestion consumes replicated snapshot state
    // - PRG_Distributed_Commit_Ingestion consumes replicated commit state
    //
    // This GVL intentionally separates:
    // runtime authority
    // transport replication
    // distributed reconciliation
    // ======================================================

    HA_Replication_Enabled : BOOL := FALSE;
    HA_Channel_Healthy : BOOL := FALSE;

    HA_Last_TX_MS : UDINT := 0;
    HA_Last_RX_MS : UDINT := 0;

    HA_Remote_Session_Valid : BOOL := FALSE;
    HA_Remote_Last_Refresh_MS : UDINT := 0;

    HA_Remote_Runtime_Epoch : ULINT := 0;
    HA_Remote_Snapshot_Epoch : ULINT := 0;
    HA_Remote_Boot_Generation : ULINT := 0;
    HA_Remote_Fencing_Token : ULINT := 0;

    HA_Remote_Publication_Allowed : BOOL := FALSE;
    HA_Remote_Runtime_Healthy : BOOL := FALSE;

    HA_Remote_Distributed_Snapshot_Epoch : ULINT := 0;
    HA_Remote_Runtime_Snapshot_Epoch : ULINT := 0;
    HA_Remote_Publication_Epoch : ULINT := 0;
    HA_Remote_Snapshot_Immutable : BOOL := FALSE;
    HA_Remote_Snapshot_Last_Refresh_MS : UDINT := 0;

    HA_Remote_Publication_Commit_Epoch : ULINT := 0;
    HA_Remote_Prepare_Epoch : ULINT := 0;
    HA_Remote_Commit_Ack_Valid : BOOL := FALSE;
    HA_Remote_Commit_Last_Refresh_MS : UDINT := 0;
END_VAR

(* ---- GVL_HEALTH_BRIDGE.gvl ---- *)
{attribute 'qualified_only'}
VAR_GLOBAL
    G_Smoke_Detected : BOOL;
    G_Gas_Detected : BOOL;
    G_Methane_Warning_Level : BOOL;
    G_Methane_Alarm_Level : BOOL;
    G_Methane_Critical_Level : BOOL;
    G_Leak_Detected : BOOL;
    G_Leak_Warning_Level : BOOL;
    G_CO_Warning_Level : BOOL;
    G_CO_Alarm_Level : BOOL;
    G_Last_Fault_Event_Text : STRING(255);
    G_Role_Conflict_Error : BOOL;
END_VAR

(* ---- GVL_Heating_Circuit_Explainability.gvl ---- *)
{attribute 'qualified_only'}
VAR_GLOBAL
    // ==============================================================================
    // Heating circuit explainability compatibility publication surface
    // ==============================================================================
    //
    // Passive compatibility/HMI/diagnostic publication layer.
    // Observation-only: no command, output or runtime authority.
    //
    // IMPORTANT ARCHITECTURAL ROLE:
    //
    // This GVL is NOT:
    // - canonical runtime ingestion;
    // - predictive routing root;
    // - supervisory aggregation root;
    // - runtime authority surface.
    //
    // Canonical routing model:
    //
    // runtime
    //   -> GVL_Heating_Runtime_Projection
    //   -> adapters/enrichment
    //   -> GVL_Heating_Runtime_Supervisory_Publication
    //   -> compatibility/HMI publication surfaces
    //
    // This GVL exists to preserve:
    // - HMI compatibility;
    // - diagnostics compatibility;
    // - historical publication continuity;
    // - migration stability.
    // ==============================================================================

    // Passive per-circuit heating source-selection explainability.
    G_Source_Selection_Visible : ARRAY[1..GVL_CONSTANTS.C_MAX_HEATING_CIRCUITS] OF BOOL;
    G_Selected_Source_Code : ARRAY[1..GVL_CONSTANTS.C_MAX_HEATING_CIRCUITS] OF UINT; // 0 none, 1 room, 2 floor
    G_Selected_Source_Text : ARRAY[1..GVL_CONSTANTS.C_MAX_HEATING_CIRCUITS] OF STRING(64);
    G_Fallback_Active : ARRAY[1..GVL_CONSTANTS.C_MAX_HEATING_CIRCUITS] OF BOOL;
    G_Source_Degraded : ARRAY[1..GVL_CONSTANTS.C_MAX_HEATING_CIRCUITS] OF BOOL;

    // Canonical source semantics live in runtime projection contracts.
    G_Selected_Source_Confidence : ARRAY[1..GVL_CONSTANTS.C_MAX_HEATING_CIRCUITS] OF REAL;

    // Compatibility mirrors only.
    G_Primary_Source_Confidence : ARRAY[1..GVL_CONSTANTS.C_MAX_HEATING_CIRCUITS] OF REAL;
    G_Fallback_Source_Confidence : ARRAY[1..GVL_CONSTANTS.C_MAX_HEATING_CIRCUITS] OF REAL;

    // Explainability publication.
    G_Reason_Code : ARRAY[1..GVL_CONSTANTS.C_MAX_HEATING_CIRCUITS] OF UINT; // 0 OK, 1 primary degraded fallback used, 2 degraded primary retained, 3 source loss
    G_Reason_Text : ARRAY[1..GVL_CONSTANTS.C_MAX_HEATING_CIRCUITS] OF STRING(128);

    // Passive edge/event publication for compatibility visibility.
    // Canonical event semantics live in runtime projection contracts.
    G_Source_Switched_Event : ARRAY[1..GVL_CONSTANTS.C_MAX_HEATING_CIRCUITS] OF BOOL;
    G_Fallback_Activated_Event : ARRAY[1..GVL_CONSTANTS.C_MAX_HEATING_CIRCUITS] OF BOOL;
    G_Fallback_Recovered_Event : ARRAY[1..GVL_CONSTANTS.C_MAX_HEATING_CIRCUITS] OF BOOL;
    G_Source_Loss_Event : ARRAY[1..GVL_CONSTANTS.C_MAX_HEATING_CIRCUITS] OF BOOL;

    G_Last_Event_MS : ARRAY[1..GVL_CONSTANTS.C_MAX_HEATING_CIRCUITS] OF UDINT;
    G_Last_Event_Code : ARRAY[1..GVL_CONSTANTS.C_MAX_HEATING_CIRCUITS] OF UINT; // 0 none, 1 switched, 2 fallback activated, 3 fallback recovered, 4 source loss
    G_Last_Event_Text : ARRAY[1..GVL_CONSTANTS.C_MAX_HEATING_CIRCUITS] OF STRING(128);
END_VAR

(* ---- GVL_HEATING_DIAGNOSTICS.gvl ---- *)
VAR_GLOBAL
    G_Manifold_Pressure_Fault : ARRAY[1..GVL_CONSTANTS.C_MAX_MANIFOLDS] OF BOOL;
    G_Manifold_Current_Fault : ARRAY[1..GVL_CONSTANTS.C_MAX_MANIFOLDS] OF BOOL;
    G_Manifold_Return_Temp_Fault : ARRAY[1..GVL_CONSTANTS.C_MAX_MANIFOLDS] OF BOOL;
END_VAR

(* ---- GVL_HEATING_DOMAIN_STATUS.gvl ---- *)
{attribute 'qualified_only'}
VAR_GLOBAL
    // Heating domain status. Observational only.

    G_Runtime_Required : BOOL := FALSE;
    G_Runtime_Executed : BOOL := FALSE;
    G_Runtime_Idle_By_Design : BOOL := FALSE;
    G_Runtime_Blocked_By_Command : BOOL := FALSE;
    G_Emergency_Stop_Active : BOOL := FALSE;
    G_Gas_Safety_Stop_Active : BOOL := FALSE;
    G_Any_Zone_Valve_Active : BOOL := FALSE;
    G_Any_Manifold_Pump_Active : BOOL := FALSE;
    G_Any_Manifold_Valve_Active : BOOL := FALSE;
    G_DHW_Active : BOOL := FALSE;
    G_Freeze_Context_Active : BOOL := FALSE;
    G_Last_Update_MS : UDINT := 0;
    G_Status_Code : UINT := 0;
    G_Status_Text : STRING(128) := '';
END_VAR

(* ---- GVL_HEATING_OUTPUT.gvl ---- *)
VAR_GLOBAL
    // Heating output projection produced by PRG_Heating and consumed by PRG_IO_Write.
    // This removes the direct PRG_IO_Write -> GVL_STATE dependency for Heating physical outputs.

    DO_Zone_Valves : ARRAY[1..8] OF BOOL;
    DO_Manifold_Pumps : ARRAY[1..GVL_CONSTANTS.C_MAX_MANIFOLDS] OF BOOL;
    AO_Manifold_Valves : ARRAY[1..GVL_CONSTANTS.C_MAX_MANIFOLDS] OF UINT;

    DO_DHW_Heating_Pump : BOOL := FALSE;
    DO_DHW_Circ_Pump : BOOL := FALSE;
    DO_Backup_Circulation_Pump : BOOL := FALSE;
    DO_Electric_Heater_Enable : BOOL := FALSE;
END_VAR

(* ---- GVL_HEATING_POLICY.gvl ---- *)
{attribute 'qualified_only'}
VAR_GLOBAL
    G_Zone_Empty_Duration_MS : ARRAY[1..GVL_CONSTANTS.C_MAX_ZONES] OF UDINT;
    G_Zone_Permanent_Use : ARRAY[1..GVL_CONSTANTS.C_MAX_ZONES] OF BOOL;
    G_Zone_Guest_Preheat_Request : ARRAY[1..GVL_CONSTANTS.C_MAX_ZONES] OF BOOL;
    G_Zone_Policy_Class : ARRAY[1..GVL_CONSTANTS.C_MAX_ZONES] OF INT;
    G_Zone_Target_Adjustment : ARRAY[1..GVL_CONSTANTS.C_MAX_ZONES] OF REAL;
    G_Zone_Priority_Bias : ARRAY[1..GVL_CONSTANTS.C_MAX_ZONES] OF REAL;

    G_Policy_Mode : E_Heating_Policy_Mode := E_Heating_Policy_Mode.HPM_NORMAL;
    G_Policy_Block_Heating_Request : BOOL;
    G_Policy_Target_Adjustment : REAL;
    G_Policy_Priority_Multiplier : REAL := 1.0;
    G_Policy_Self_Tune_Active : BOOL;
    G_Policy_Self_Tune_Level : INT;
    G_Policy_Feedback_Stable : BOOL;
    G_Policy_Feedback_Improving : BOOL;
    G_Policy_Feedback_Quality : REAL;
    G_Policy_Predictive_Active : BOOL;
    G_Policy_Predictive_Adjustment : REAL;

    // zone intelligence
    G_Zone_Quality : ARRAY[1..GVL_CONSTANTS.C_MAX_ZONES] OF REAL;
    G_Zone_Improving : ARRAY[1..GVL_CONSTANTS.C_MAX_ZONES] OF BOOL;
    G_Zone_Stable : ARRAY[1..GVL_CONSTANTS.C_MAX_ZONES] OF BOOL;
    G_Zone_Self_Level : ARRAY[1..GVL_CONSTANTS.C_MAX_ZONES] OF INT;

    // thermal model: 1.0 = normal inertia, >1 slower/heavier, <1 faster/lighter
    G_Zone_Thermal_Inertia : ARRAY[1..GVL_CONSTANTS.C_MAX_ZONES] OF REAL := [1.0, 1.0, 1.0, 1.0, 1.0, 1.0, 1.0, 1.0, 1.0, 1.0, 1.0, 1.0, 1.0, 1.0, 1.0, 1.0];
    G_Zone_Thermal_Response : ARRAY[1..GVL_CONSTANTS.C_MAX_ZONES] OF REAL;
    G_Zone_Thermal_Demand : ARRAY[1..GVL_CONSTANTS.C_MAX_ZONES] OF REAL;
    G_Zone_Time_To_Heat_MS : ARRAY[1..GVL_CONSTANTS.C_MAX_ZONES] OF UDINT;
    G_Zone_Preheat_Needed : ARRAY[1..GVL_CONSTANTS.C_MAX_ZONES] OF BOOL;

    // thermal model v2 diagnostics
    G_Zone_Heat_Loss_Rate : ARRAY[1..GVL_CONSTANTS.C_MAX_ZONES] OF REAL;
    G_Zone_Heat_Gain_Rate : ARRAY[1..GVL_CONSTANTS.C_MAX_ZONES] OF REAL;
    G_Zone_Predicted_Temp_30m : ARRAY[1..GVL_CONSTANTS.C_MAX_ZONES] OF REAL;
    G_Zone_Thermal_Model_Confidence : ARRAY[1..GVL_CONSTANTS.C_MAX_ZONES] OF REAL;

    // schedule-aware preheat. Comfort time is milliseconds from midnight.
    G_Zone_Schedule_Enabled : ARRAY[1..GVL_CONSTANTS.C_MAX_ZONES] OF BOOL;
    G_Zone_Comfort_Time_MS : ARRAY[1..GVL_CONSTANTS.C_MAX_ZONES] OF UDINT;
    G_Zone_Schedule_Preheat_Active : ARRAY[1..GVL_CONSTANTS.C_MAX_ZONES] OF BOOL;
    G_Zone_Schedule_Learned_Offset_MS : ARRAY[1..GVL_CONSTANTS.C_MAX_ZONES, 1..3] OF UDINT;
END_VAR

(* ---- GVL_HEATING_POLICY_CONFIG.gvl ---- *)
{attribute 'qualified_only'}
VAR_GLOBAL
    G_Guest_Preheat_Enabled : BOOL := TRUE;
    G_Guest_Preheat_Priority_Boost : INT := 2;
    G_Guest_Preheat_Max_Duration_MS : UDINT := 7200000;

    // HMI-configurable schedule (per zone, up to 3 events)
    G_Zone_Schedule : ARRAY[1..GVL_CONSTANTS.C_MAX_ZONES, 1..3] OF ST_Heating_Schedule_Event;
END_VAR

(* ---- GVL_HEATING_REQUEST.st ---- *)
VAR_GLOBAL
    G_Preheat_Request : BOOL := FALSE;
END_VAR

(* ---- GVL_Heating_Runtime_Explainability.gvl ---- *)
{attribute 'qualified_only'}
VAR_GLOBAL
    // Passive runtime explainability publication surface.
    // Observation-only: no command, output or runtime authority.
    G_Runtime_Phase_Event : ST_Heating_Runtime_Phase_Event;
    G_Runtime_Anomaly : ST_Heating_Runtime_Anomaly;
    G_Runtime_Blackbox_Event : ST_Heating_Runtime_Blackbox_Event;
    G_Runtime_Adaptive_Intelligence : ST_Heating_Runtime_Adaptive_Intelligence;
    G_Runtime_Causality_Graph : ST_Heating_Runtime_Causality_Graph;
    G_Runtime_Integration_Bridge : ST_Heating_Runtime_Integration_Bridge;
    G_Runtime_Predictive_State : ST_Heating_Runtime_Predictive_State;
    G_Runtime_Execution_Timeline : ST_Heating_Runtime_Execution_Timeline;
    G_Runtime_Phase_Transition : ST_Heating_Runtime_Phase_Transition;

    G_Runtime_Explainability_Publication_Valid : BOOL := FALSE;
    G_Runtime_Explainability_Status_Code : UINT := 0;
    G_Runtime_Explainability_Status_Text : STRING(128) := 'Heating runtime explainability inactive';
END_VAR

(* ---- GVL_Heating_Runtime_Meta.gvl ---- *)
{attribute 'qualified_only'}
VAR_GLOBAL
    // Passive runtime meta-supervision publication surface.
    // Observation-only: no command, output or runtime authority.
    G_Runtime_Meta_Supervision : ST_Heating_Runtime_Meta_Supervision;
    G_Runtime_Meta_Publication_Valid : BOOL := FALSE;
    G_Runtime_Meta_Status_Code : UINT := 0;
    G_Runtime_Meta_Status_Text : STRING(128) := 'Heating runtime meta supervision inactive';
END_VAR

(* ---- GVL_Heating_Runtime_Observation.gvl ---- *)
VAR_GLOBAL
    G_Runtime_Observer_Lifecycle_State : E_Runtime_Observer_Lifecycle_State := E_Runtime_Observer_Lifecycle_State.ROS_INACTIVE;
    G_Runtime_Observer_Lifecycle_Code : UINT := 0;
    G_Runtime_Observer_Lifecycle_Text : STRING(128) := 'Heating runtime observer inactive';
    G_Runtime_Observer_Commissioning_Required : BOOL := TRUE;
    G_Runtime_Observer_Commissioning_Active : BOOL := FALSE;
    G_Runtime_Observer_Commissioning_Complete : BOOL := FALSE;
    G_Runtime_Observation : ST_Heating_Runtime_Observation;
    G_Runtime_Observation_Publication_Valid : BOOL := FALSE;
    G_Runtime_Observation_Stabilization_Complete : BOOL := FALSE;
    G_Runtime_Observation_Operational : BOOL := FALSE;
    G_Runtime_Observation_Valid : BOOL := FALSE;
    G_Runtime_Observer_Ready : BOOL := FALSE;
    G_Runtime_Observer_Fault : BOOL := FALSE;
    G_Runtime_Observation_Status_Code : UINT := 0;
    G_Runtime_Observation_Status_Text : STRING(128) := 'Heating runtime observation inactive';
END_VAR

(* ---- GVL_Heating_Runtime_Observer.gvl ---- *)
VAR_GLOBAL
    G_Runtime_Observer_Lifecycle_State : E_Runtime_Observer_Lifecycle_State := E_Runtime_Observer_Lifecycle_State.ROS_INACTIVE;
    G_Runtime_Observer_Enable_Request : BOOL := FALSE;
    G_Runtime_Observer_Enable_Authorized : BOOL := FALSE;
    G_Runtime_Observer_Enable_Effective : BOOL := FALSE;
    G_Runtime_Observer_Bootstrap_Mode : BOOL := TRUE;
    G_Runtime_Observer_Passive_Mode : BOOL := TRUE;
    G_Runtime_Observer_ReadOnly_Mode : BOOL := TRUE;
    G_Runtime_Observer_Activation_Validated : BOOL := FALSE;
    G_Runtime_Observer_Sequencing_Validated : BOOL := FALSE;
    G_Runtime_Observer_Publication_Validated : BOOL := FALSE;
    G_Runtime_Observer_Rollback_Validated : BOOL := FALSE;
    G_Runtime_Observer_Governance_Locked : BOOL := TRUE;
    G_Runtime_Observer_Runtime_Authority_Disabled : BOOL := TRUE;
    G_Runtime_Observer_Writable_Exports_Disabled : BOOL := TRUE;
    G_Runtime_Observer_Predictive_Disabled : BOOL := TRUE;
    G_Runtime_Observer_Adaptive_Disabled : BOOL := TRUE;
    G_Runtime_Observer_Replay_Disabled : BOOL := TRUE;

    G_Runtime_Observer_Authorization_Valid : BOOL := FALSE;

    G_Runtime_Observer_Authorization_Status_Code : UINT := 0;
    G_Runtime_Observer_Authorization_Status_Text : STRING(128) := 'Heating runtime observer authorization inactive';
END_VAR

(* ---- GVL_Heating_Runtime_Projection.gvl ---- *)
{attribute 'qualified_only'}
VAR_GLOBAL
    // Canonical passive runtime projection surface.
    // Runtime publishes semantic state only.
    // Supervisory layers may observe but never control through this surface.

    G_Circuit_Projection : ARRAY[1..GVL_CONSTANTS.C_MAX_HEATING_CIRCUITS] OF ST_Heating_Circuit_Runtime_Projection;
END_VAR

(* ---- GVL_Heating_Source_Stability.gvl ---- *)
{attribute 'qualified_only'}
VAR_GLOBAL
    // Predictive source-stability observability layer.
    // Observation-only: no runtime authority, no valve ownership,
    // no direct influence on heating outputs.

    G_Stability_Visible : ARRAY[1..GVL_CONSTANTS.C_MAX_HEATING_CIRCUITS] OF BOOL;

    // Oscillation / switching observation
    G_Source_Switch_Count : ARRAY[1..GVL_CONSTANTS.C_MAX_HEATING_CIRCUITS] OF UINT;
    G_Fallback_Activation_Count : ARRAY[1..GVL_CONSTANTS.C_MAX_HEATING_CIRCUITS] OF UINT;
    G_Fallback_Recovery_Count : ARRAY[1..GVL_CONSTANTS.C_MAX_HEATING_CIRCUITS] OF UINT;
    G_Source_Loss_Count : ARRAY[1..GVL_CONSTANTS.C_MAX_HEATING_CIRCUITS] OF UINT;

    // Trend / persistence observation
    G_Degraded_Trend_Visible : ARRAY[1..GVL_CONSTANTS.C_MAX_HEATING_CIRCUITS] OF BOOL;
    G_Recovery_Trend_Visible : ARRAY[1..GVL_CONSTANTS.C_MAX_HEATING_CIRCUITS] OF BOOL;
    G_Oscillation_Detected : ARRAY[1..GVL_CONSTANTS.C_MAX_HEATING_CIRCUITS] OF BOOL;
    G_Instability_Attention : ARRAY[1..GVL_CONSTANTS.C_MAX_HEATING_CIRCUITS] OF BOOL;

    // Predictive scoring
    G_Instability_Score : ARRAY[1..GVL_CONSTANTS.C_MAX_HEATING_CIRCUITS] OF REAL;
    G_Confidence_Volatility : ARRAY[1..GVL_CONSTANTS.C_MAX_HEATING_CIRCUITS] OF REAL;
    G_Source_Trust_Trend : ARRAY[1..GVL_CONSTANTS.C_MAX_HEATING_CIRCUITS] OF REAL;

    // Explainability publication
    G_Status_Code : ARRAY[1..GVL_CONSTANTS.C_MAX_HEATING_CIRCUITS] OF UINT;
    G_Status_Text : ARRAY[1..GVL_CONSTANTS.C_MAX_HEATING_CIRCUITS] OF STRING(128);
    G_Last_Observation_MS : ARRAY[1..GVL_CONSTANTS.C_MAX_HEATING_CIRCUITS] OF UDINT;
END_VAR

(* ---- GVL_HMI.gvl ---- *)
{attribute 'qualified_only'}
VAR_GLOBAL
    // Heating dashboard
    G_HMI_Heating_Confidence : REAL := 1.0;
    G_HMI_Heating_Confidence_Percent : INT := 100;
    G_HMI_Heating_Reason_Code : INT := 0;
    G_HMI_Heating_Status_Text : STRING(128) := 'OK';
    G_HMI_Heating_Status_Level : INT := 0; // 0=OK, 1=WARN, 2=ALARM

    // Heating cascade dashboard
    G_HMI_Heating_Cascade_Available : BOOL;
    G_HMI_Heating_Cascade_Degraded : BOOL;
    G_HMI_Heating_Cascade_Partial_Capacity : BOOL;
    G_HMI_Heating_Cascade_No_Flame : BOOL;
    G_HMI_Heating_Cascade_Transport_Degraded : BOOL;
    G_HMI_Heating_Cascade_Ignition_Timeout : BOOL;
    G_HMI_Heating_Cascade_Active_Boilers : UINT;
    G_HMI_Heating_Cascade_Available_Boilers : UINT;

    // OpenTherm dashboard
    G_HMI_Boiler_OT_Online : ARRAY[1..GVL_CONSTANTS.C_MAX_BOILERS] OF BOOL;
    G_HMI_Boiler_OT_Command_Ack : ARRAY[1..GVL_CONSTANTS.C_MAX_BOILERS] OF BOOL;
    G_HMI_Boiler_OT_Command_Timeout : ARRAY[1..GVL_CONSTANTS.C_MAX_BOILERS] OF BOOL;
    G_HMI_Boiler_OT_Heartbeat_Timeout : ARRAY[1..GVL_CONSTANTS.C_MAX_BOILERS] OF BOOL;
    G_HMI_Boiler_OT_Adapter_Error : ARRAY[1..GVL_CONSTANTS.C_MAX_BOILERS] OF BOOL;
    G_HMI_Boiler_OT_Heartbeat_Age_MS : ARRAY[1..GVL_CONSTANTS.C_MAX_BOILERS] OF UDINT;
    G_HMI_Boiler_OT_Command_Age_MS : ARRAY[1..GVL_CONSTANTS.C_MAX_BOILERS] OF UDINT;
    G_HMI_Boiler_OT_Adapter_State : ARRAY[1..GVL_CONSTANTS.C_MAX_BOILERS] OF E_OpenTherm_Adapter_State;
    G_HMI_Boiler_OT_Error_State : ARRAY[1..GVL_CONSTANTS.C_MAX_BOILERS] OF E_OpenTherm_Error;

    // Heating predictive dashboard
    G_HMI_Heating_Predictive_Pressure_Drop : ARRAY[1..GVL_CONSTANTS.C_MAX_MANIFOLDS] OF BOOL;
    G_HMI_Heating_Predictive_Current_Rise : ARRAY[1..GVL_CONSTANTS.C_MAX_MANIFOLDS] OF BOOL;

    // File/archive dashboard. Read-only projection of GVL_FILE_ARCHIVE status.
    // HMI requests still go through GVL_FILE_ARCHIVE one-shot request fields.
    G_HMI_File_Archive_Interface_Enabled : BOOL;
    G_HMI_File_Archive_CSV_Enabled : BOOL;
    G_HMI_File_Archive_Target_Code : BYTE;
    G_HMI_File_Archive_Target_Available : BOOL;
    G_HMI_File_Archive_Write_Busy : BOOL;
    G_HMI_File_Archive_Write_Done : BOOL;
    G_HMI_File_Archive_Write_Error : BOOL;
    G_HMI_File_Archive_Last_Error_Code : UDINT;
    G_HMI_File_Archive_Last_Status_Text : STRING(200);
    G_HMI_File_Archive_Last_Write_MS : UDINT;
    G_HMI_File_Archive_Status_Level : INT := 0; // 0=OK, 1=WARN, 2=ERROR

    // Automatic config backup dashboard.
    G_HMI_File_Archive_Auto_Backup_Enabled : BOOL;
    G_HMI_File_Archive_Auto_Backup_Time_Of_Day_MS : UDINT;
    G_HMI_File_Archive_Auto_Backup_Last_Day_Of_Week : INT;
    G_HMI_File_Archive_Auto_Backup_Last_Request_MS : UDINT;
    G_HMI_File_Archive_Auto_Backup_Last_Status_Text : STRING(200);

    // Water emergency-open dashboard. Read-only projection of emergency access state.
    G_HMI_Water_Emergency_Open_Active : ARRAY[1..4] OF BOOL;
    G_HMI_Water_Emergency_Open_Remaining_MS : ARRAY[1..4] OF UDINT;
    G_HMI_Water_Emergency_Open_Count_Today : ARRAY[1..4] OF INT;
    G_HMI_Water_Emergency_Open_Any_Active : BOOL;
    G_HMI_Water_Emergency_Open_Last_Accepted : BOOL;
    G_HMI_Water_Emergency_Open_Last_Denied : BOOL;
    G_HMI_Water_Emergency_Open_Last_Denial_Code : UINT;
    G_HMI_Water_Emergency_Open_Last_Event_Group : INT;
    G_HMI_Water_Emergency_Open_Last_Event_MS : UDINT;
    G_HMI_Water_Emergency_Open_Status_Text : STRING(200);
    G_HMI_Water_Emergency_Open_Status_Level : INT := 0; // 0=OK, 1=ACTIVE, 2=DENIED

    // Water valve diagnostics dashboard. Logical valves 1..6 local, 7=35, 8=36.
    G_HMI_Water_Valve_Command_Open : ARRAY[1..8] OF BOOL;
    G_HMI_Water_Valve_Command_Close : ARRAY[1..8] OF BOOL;
    G_HMI_Water_Valve_Open_FB : ARRAY[1..8] OF BOOL;
    G_HMI_Water_Valve_Close_FB : ARRAY[1..8] OF BOOL;
    G_HMI_Water_Valve_Movement_Timeout_MS : ARRAY[1..8] OF UDINT;
    G_HMI_Water_Valve_Open_Fault : ARRAY[1..8] OF BOOL;
    G_HMI_Water_Valve_Close_Fault : ARRAY[1..8] OF BOOL;
    G_HMI_Water_Valve_Critical_Close_Fault : ARRAY[1..8] OF BOOL;
    G_HMI_Water_Valve_Open_Blocked : ARRAY[1..8] OF BOOL;
    G_HMI_Water_Valve_Open_Block_Active : BOOL;
    G_HMI_Water_Valve_Open_Block_Text : STRING(200);
    G_HMI_Water_Valve_Service_Last_Reset_Accepted : BOOL;
    G_HMI_Water_Valve_Service_Last_Reset_Denied : BOOL;
    G_HMI_Water_Valve_Service_Last_Reset_Denial_Code : UINT;
    G_HMI_Water_Valve_Service_Last_Reset_Valve_Index : INT;
    G_HMI_Water_Valve_Service_Last_Reset_MS : UDINT;
    G_HMI_Water_Valve_Service_Status_Text : STRING(200);
    G_HMI_Water_Valve_Close_Fault_Active : BOOL;
    G_HMI_Water_Valve_Main_Shutdown_Recommended : BOOL;
    G_HMI_Water_Valve_Localization_Failed : BOOL;
    G_HMI_Water_Valve_Close_Fault_Text : STRING(200);
    G_HMI_Water_Valve_Escalation_Text : STRING(200);
    G_HMI_Water_Valve_Status_Level : INT := 0; // 0=OK, 1=WARN, 2=CRITICAL

    // Config control dashboard. Read-only projection of staged apply and rollback state.
    G_HMI_Config_Control_Version : UDINT;
    G_HMI_Config_Control_Last_Good_Version : UDINT;
    G_HMI_Config_Control_Staged_Config_Version : UDINT;
    G_HMI_Config_Control_Staged_Last_Changed_MS : UDINT;
    G_HMI_Config_Control_Backup_Valid : BOOL;
    G_HMI_Config_Control_Apply_Pending : BOOL;
    G_HMI_Config_Control_Rollback_Pending : BOOL;
    G_HMI_Config_Control_Apply_Done : BOOL;
    G_HMI_Config_Control_Rollback_Done : BOOL;
    G_HMI_Config_Control_Reset_Default_Done : BOOL;
    G_HMI_Config_Control_Config_Valid : BOOL;
    G_HMI_Config_Control_Last_Action_Text : STRING(128);
    G_HMI_Config_Control_Last_Error_Text : STRING(200);
    G_HMI_Config_Control_Last_Update_MS : UDINT;
    G_HMI_Config_Control_Status_Level : INT := 0; // 0=OK, 1=WARN, 2=ERROR

    // Config workflow dashboard.
    G_HMI_Config_Workflow_Runtime_Valid : BOOL;
    G_HMI_Config_Workflow_Draft_Dirty : BOOL;
    G_HMI_Config_Workflow_Validation_OK : BOOL;
    G_HMI_Config_Workflow_Validation_Failed : BOOL;
    G_HMI_Config_Workflow_Draft_Version : UDINT;
    G_HMI_Config_Workflow_Validated_Draft_Version : UDINT;
    G_HMI_Config_Workflow_Topology_Draft_Version : UDINT;
    G_HMI_Config_Workflow_Validated_Topology_Version : UDINT;
    G_HMI_Config_Workflow_Validation_Last_Run_MS : UDINT;
    G_HMI_Config_Workflow_Validation_Result_Seq : UDINT;
    G_HMI_Config_Workflow_Topology_Activation_Required : BOOL;
    G_HMI_Config_Workflow_Topology_Validation_OK : BOOL;
    G_HMI_Config_Workflow_Status_Code : UINT;
    G_HMI_Config_Workflow_Status_Text : STRING(160);
    G_HMI_Config_Workflow_Status_Level : INT := 0; // 0=OK, 1=WARN, 2=ERROR

    // Config simulation dashboard.
    G_HMI_Config_Simulation_Request_Pending : BOOL;
    G_HMI_Config_Simulation_Result_OK : BOOL;
    G_HMI_Config_Simulation_Error_Text : STRING(200);
    G_HMI_Config_Simulation_Last_Run_MS : UDINT;
    G_HMI_Config_Simulation_Result_Seq : UDINT;
    G_HMI_Config_Simulation_Staged_Config_Version : UDINT;
    G_HMI_Config_Simulation_Status_Level : INT := 0; // 0=OK, 1=PENDING, 2=ERROR
END_VAR

(* ---- GVL_HMI_ACCESS.gvl ---- *)
{attribute 'qualified_only'}
VAR_GLOBAL
    G_Safety_Mode : E_Safety_Mode := NORMAL;
    G_User_Access_Level : INT := 0;
    G_Manual_Access_OK : BOOL := FALSE;

    G_Runtime_Required : BOOL;
    G_Runtime_Executed : BOOL;
    G_Runtime_Idle_By_Design : BOOL;
    G_Runtime_Blocked_By_Distributed_Gates : BOOL;
    G_Any_Pulse_Active : BOOL;
    G_Last_Update_MS : UDINT;
    G_Status_Code : UINT;
    G_Status_Text : STRING(128);

    G_Command_Lock_1_Open : BOOL;
    G_Command_Lock_1_Close : BOOL;
    G_Command_Lock_2_Open : BOOL;
    G_Command_Lock_2_Close : BOOL;
    G_Command_Gate_Open : BOOL;
    G_Command_Wicket_Open : BOOL;

    G_Output_Lock_1_Open : BOOL;
    G_Output_Lock_1_Close : BOOL;
    G_Output_Lock_2_Open : BOOL;
    G_Output_Lock_2_Close : BOOL;
    G_Output_Gate_Open : BOOL;
    G_Output_Wicket_Open : BOOL;

    G_Physical_Lock_1_Open : BOOL;
    G_Physical_Lock_1_Close : BOOL;
    G_Physical_Lock_2_Open : BOOL;
    G_Physical_Lock_2_Close : BOOL;
    G_Physical_Gate_Open : BOOL;
    G_Physical_Wicket_Open : BOOL;

    G_Fire_Evacuation_Access_Active : BOOL;
    G_Gas_Access_Release_Active : BOOL;
    G_Safety_Cleared_Active : BOOL;
    G_Distributed_Block_Active : BOOL;
    G_Reason_Text : STRING(160);
END_VAR

(* ---- GVL_HMI_ALARM_AUDIBLE_ACK.gvl ---- *)
{attribute 'qualified_only'}
VAR_GLOBAL
    G_Ack_Active : BOOL;
    G_Ack_Remaining_MS : UDINT;
    G_Ack_Count_Current_Alarm : INT;
    G_Ack_Limit_Reached : BOOL;
    G_Last_Ack_Accepted : BOOL;
    G_Last_Ack_Denied : BOOL;
    G_Last_Denial_Code : UINT;
    G_Last_Event_MS : UDINT;
    G_Status_Text : STRING(200);
    G_Effective_Siren_Muted : BOOL;

    G_Global_Siren_Request : BOOL;
    G_Global_Critical : BOOL;
    G_Gas_Fire_Siren_Request : BOOL;
    G_Security_Siren_Request : BOOL;
    G_Output_Gas_Siren : BOOL;
    G_Output_Fire_Siren : BOOL;
    G_Output_Security_Siren : BOOL;
END_VAR

(* ---- GVL_HMI_Config_Workflow.gvl ---- *)
{attribute 'qualified_only'}
VAR_GLOBAL
    G_Open_Editor_Request : BOOL;
    G_Validate_Request : BOOL;
    G_Activate_Request : BOOL;
    G_Rollback_Request : BOOL;
    G_Reset_Default_Request : BOOL;

    G_Service_Mode_Active : BOOL;
    G_Operator_Ack : BOOL;

    G_Workflow_State : ST_HMI_Config_Workflow_State;

    G_Runtime_Valid : BOOL;
    G_Last_Update_MS : UDINT;

    G_Status_Code : UINT;
    G_Status_Text : STRING(160);
END_VAR

(* ---- GVL_HMI_GAS_SMOKE_CO.gvl ---- *)
{attribute 'qualified_only'}
VAR_GLOBAL
    G_Methane_Effective : ARRAY[1..GVL_CONSTANTS.C_MAX_METHANE_SENSORS] OF REAL;
    G_Methane_Max_LEL : REAL;
    G_Methane_Min_LEL : REAL;
    G_Methane_Diff_LEL : REAL;
    G_Methane_Max_Sensor_Index : INT;
    G_Methane_Disagreement_Active : BOOL;
    G_Methane_Disagreement_Limit_LEL : REAL;
    G_Methane_Redundancy_Available : BOOL;
    G_Methane_Conservative_Max_Selected : BOOL;
    G_Methane_Redundancy_Status_Text : STRING(160);
    G_Methane_Redundancy_Last_Update_MS : UDINT;
    G_Methane_Warning_Level : BOOL;
    G_Methane_Alarm_Level : BOOL;
    G_Methane_Critical_Level : BOOL;

    G_CO_Effective : ARRAY[1..GVL_CONSTANTS.C_MAX_CO_SENSORS] OF REAL;
    G_CO_Max_PPM : REAL;
    G_CO_Max_Sensor_Index : INT;
    G_CO_Level_30ppm_Active : BOOL;
    G_CO_Level_70ppm_Active : BOOL;
    G_CO_Level_400ppm_Active : BOOL;
    G_CO_Timer_30ppm_ET : TIME;
    G_CO_Timer_70ppm_ET : TIME;
    G_CO_Timer_400ppm_ET : TIME;
    G_CO_Timer_30ppm_Q : BOOL;
    G_CO_Timer_70ppm_Q : BOOL;
    G_CO_Timer_400ppm_Q : BOOL;
    G_CO_Exposure_Status_Text : STRING(160);
    G_CO_Exposure_Last_Update_MS : UDINT;
    G_CO_Warning_Level : BOOL;
    G_CO_Alarm_Level : BOOL;

    G_Smoke_Effective : ARRAY[1..GVL_CONSTANTS.C_MAX_SMOKE_SENSORS] OF BOOL;
    G_Smoke_Active_Count : UINT;
    G_Smoke_Detected : BOOL;
    G_Smoke_Any_Input_Active : BOOL;
    G_Smoke_Group_Active : ARRAY[1..3] OF BOOL;
    G_Smoke_Group_Pair_Confirmed : ARRAY[1..3] OF BOOL;
    G_Smoke_Group_Timer_Confirmed : ARRAY[1..3] OF BOOL;
    G_Smoke_Verified_By_Pair : BOOL;
    G_Smoke_Verified_By_Timer : BOOL;
    G_Smoke_Verified_Group : INT;
    G_Smoke_Verification_Text : STRING(160);
    G_Smoke_Verification_Last_Update_MS : UDINT;
    G_Smoke_Exhaust_Targeted : BOOL;
    G_Smoke_Exhaust_Fallback_All : BOOL;
    G_Smoke_Exhaust_Target_Group : INT;
    G_Smoke_Target_Exhaust_Fans : ARRAY[1..GVL_CONSTANTS.C_MAX_EXHAUST_FANS] OF BOOL;

    G_Gas_Detected : BOOL;
    G_Status_Text : STRING(200);
    G_Status_Level : INT := 0; // 0=OK, 1=WARN, 2=ALARM, 3=CRITICAL

    G_Safety_Fire_Alarm_Active : BOOL;
    G_Safety_Gas_Alarm_Active : BOOL;
    G_Safety_CO_Warning_Active : BOOL;
    G_Gas_Close_Required : BOOL;
    G_Boiler_Stop_Required : BOOL;
    G_System_Safe_Stop_Required : BOOL;
    G_Evacuation_Mode_Active : BOOL;
    G_Vent_Stop_Required : BOOL;
    G_Vent_Force_PV3_Boost : BOOL;
    G_Vent_Force_Supply_100 : BOOL;
    G_Vent_Force_Supply_80 : BOOL;
    G_Vent_Force_Exhaust_100 : BOOL;

    G_Command_Gas_Valve_Close : BOOL;
    G_Command_Boiler_Stop : BOOL;
    G_Output_Gas_Valve_Close : BOOL;

    G_OpenTherm_Command_Enable : ARRAY[1..GVL_CONSTANTS.C_MAX_BOILERS] OF BOOL;
    G_OpenTherm_Command_Setpoint_x10 : ARRAY[1..GVL_CONSTANTS.C_MAX_BOILERS] OF UINT;
    G_OpenTherm_Command_Sequence : ARRAY[1..GVL_CONSTANTS.C_MAX_BOILERS] OF UDINT;
    G_OpenTherm_Wire_Enable : ARRAY[1..GVL_CONSTANTS.C_MAX_BOILERS] OF WORD;
    G_OpenTherm_Wire_Setpoint_x10 : ARRAY[1..GVL_CONSTANTS.C_MAX_BOILERS] OF UINT;

    G_Vent_Output_Enable : BOOL;
    G_Vent_Output_Supply_Fans : ARRAY[1..GVL_CONSTANTS.C_MAX_SUPPLY_FANS] OF UINT;
    G_Vent_Output_Exhaust_Fans : ARRAY[1..GVL_CONSTANTS.C_MAX_EXHAUST_FANS] OF UINT;
END_VAR

(* ---- GVL_HMI_SECURITY.gvl ---- *)
{attribute 'qualified_only'}
VAR_GLOBAL
    G_Armed : BOOL;
    G_Alarm_Active : BOOL;
    G_Siren_Request : BOOL;
    G_Security_Alarm : BOOL;
    G_Security_Siren : BOOL;
    G_Global_Siren : BOOL;
    G_Status_Text : STRING(200);
    G_Status_Level : INT := 0; // 0=OK, 1=ARMED, 2=ENTRY_DELAY, 3=ALARM

    G_Safety_Access_Active : BOOL;
    G_Sensor_Path_Suppressed_By_Safety : BOOL;
    G_Sensor_Path_Status_Text : STRING(160);

    G_Arming_In_Progress : BOOL;
    G_Arm_Delay_ET : TIME;
    G_Arm_Delay_Q : BOOL;
    G_Pin_Entry_Active : BOOL;
    G_Entry_Delay_ET : TIME;
    G_Entry_Delay_Q : BOOL;
    G_Pin_Fail_Count : BYTE;
    G_Max_Attempts : BYTE;
    G_Disarm_Pending : BOOL;
    G_2FA_Required : BOOL;
    G_2FA_Send_Code_Req : BOOL;
    G_Combined_Window_Active : BOOL;
    G_Combined_Event_Count : INT;
    G_Perimeter_Active_Count : INT;
    G_Perimeter_Event_Count : INT;
    G_Any_Sensor_Active : BOOL;
    G_Door_Blocking_Open : BOOL;
    G_Window_Blocking_Open : BOOL;
    G_Workflow_Status_Text : STRING(200);
    G_Workflow_Last_Update_MS : UDINT;

    G_Motion_Active : ARRAY[1..16] OF BOOL;
    G_Door_Active : ARRAY[1..GVL_CONSTANTS.C_MAX_DOOR_SENSORS] OF BOOL;
    G_Window_Active : ARRAY[1..16] OF BOOL;

    G_Motion_Bypass : ARRAY[1..16] OF BOOL;
    G_Door_Bypass : ARRAY[1..GVL_CONSTANTS.C_MAX_DOOR_SENSORS] OF BOOL;
    G_Window_Bypass : ARRAY[1..16] OF BOOL;

    G_Motion_Active_Count : INT;
    G_Door_Active_Count : INT;
    G_Window_Active_Count : INT;
    G_Total_Active_Count : INT;

    G_Arm_Request : BOOL;
    G_Disarm_Request : BOOL;
    G_Send_2FA_Req : BOOL;
    G_Last_Update_MS : UDINT;
END_VAR

(* ---- GVL_HMI_SECURITY_ACCESS_INTENT.gvl ---- *)
{attribute 'qualified_only'}
VAR_GLOBAL
    G_Close_Request : BOOL;
    G_Close_Accepted : BOOL;
    G_Last_Request_MS : UDINT;
    G_Status_Text : STRING(160);
END_VAR

(* ---- GVL_HMI_SECURITY_IO_MAP.gvl ---- *)
{attribute 'qualified_only'}
VAR_GLOBAL
    G_Door_Map : ARRAY[1..GVL_CONSTANTS.C_MAX_DOOR_SENSORS] OF INT;
    G_Door_Map_Valid : ARRAY[1..GVL_CONSTANTS.C_MAX_DOOR_SENSORS] OF BOOL;
    G_Door_Raw_Open : ARRAY[1..GVL_CONSTANTS.C_MAX_DOOR_SENSORS] OF BOOL;

    G_Window_Map : ARRAY[1..GVL_CONSTANTS.C_MAX_ZONES] OF INT;
    G_Window_Map_Valid : ARRAY[1..GVL_CONSTANTS.C_MAX_ZONES] OF BOOL;
    G_Window_Uses_Open_Input : ARRAY[1..GVL_CONSTANTS.C_MAX_ZONES] OF BOOL;
    G_Window_Uses_Glass_Input : ARRAY[1..GVL_CONSTANTS.C_MAX_ZONES] OF BOOL;
    G_Window_Overridden_By_2F_Group : ARRAY[1..GVL_CONSTANTS.C_MAX_ZONES] OF BOOL;
    G_Window_Raw_Open : ARRAY[1..GVL_CONSTANTS.C_MAX_ZONES] OF BOOL;

    G_Group_2F_Active : BOOL;
    G_Any_Invalid_Map : BOOL;
    G_Status_Text : STRING(200);
END_VAR

(* ---- GVL_HMI_WATER_TOPOLOGY.gvl ---- *)
{attribute 'qualified_only'}
VAR_GLOBAL
    G_Active_Config_Version : UDINT;
    G_Config_Loaded : BOOL;
    G_Runtime_Valid : BOOL;
    G_Runtime_Remap_Ready : BOOL;
    G_Any_Invalid_Config : BOOL;
    G_Any_Multi_Valve_Required : BOOL;
    G_Status_Code : UINT;
    G_Status_Text : STRING(128);

    G_Sensor_Config_Valid : ARRAY[1..GVL_CONSTANTS.C_MAX_FLOOD_SENSORS] OF BOOL;
    G_Sensor_Id : ARRAY[1..GVL_CONSTANTS.C_MAX_FLOOD_SENSORS] OF UINT;
    G_Logical_Zone_Id : ARRAY[1..GVL_CONSTANTS.C_MAX_FLOOD_SENSORS] OF UINT;
    G_Hydraulic_Segment_Id : ARRAY[1..GVL_CONSTANTS.C_MAX_FLOOD_SENSORS] OF UINT;
    G_Isolation_Group_Id : ARRAY[1..GVL_CONSTANTS.C_MAX_FLOOD_SENSORS] OF UINT;
    G_Primary_Valve_Group_Id : ARRAY[1..GVL_CONSTANTS.C_MAX_FLOOD_SENSORS] OF UINT;
    G_Secondary_Valve_Group_Id : ARRAY[1..GVL_CONSTANTS.C_MAX_FLOOD_SENSORS] OF UINT;
    G_Fallback_Domain_Id : ARRAY[1..GVL_CONSTANTS.C_MAX_FLOOD_SENSORS] OF UINT;
    G_Recovery_Domain_Id : ARRAY[1..GVL_CONSTANTS.C_MAX_FLOOD_SENSORS] OF UINT;
    G_Shared_Trunk : ARRAY[1..GVL_CONSTANTS.C_MAX_FLOOD_SENSORS] OF BOOL;
    G_Cross_Zone_Dependency : ARRAY[1..GVL_CONSTANTS.C_MAX_FLOOD_SENSORS] OF BOOL;
    G_Multi_Valve_Required : ARRAY[1..GVL_CONSTANTS.C_MAX_FLOOD_SENSORS] OF BOOL;
    G_Topology_Text : ARRAY[1..GVL_CONSTANTS.C_MAX_FLOOD_SENSORS] OF STRING(160);
    G_Record_Status_Text : ARRAY[1..GVL_CONSTANTS.C_MAX_FLOOD_SENSORS] OF STRING(128);
END_VAR

(* ---- GVL_INPUT.gvl ---- *)
VAR_GLOBAL
    IN_Last_Update_MS : UDINT := 0;
    IN_Source_Valid : BOOL := FALSE;

    IN_Room_Temps : ARRAY[1..GVL_CONSTANTS.C_MAX_ZONES] OF REAL;
    IN_Floor_Temps : ARRAY[1..GVL_CONSTANTS.C_MAX_ZONES] OF REAL;
    IN_Room_Hum : ARRAY[1..GVL_CONSTANTS.C_MAX_ZONES] OF REAL;
    IN_Room_CO2 : ARRAY[1..GVL_CONSTANTS.C_MAX_ZONES] OF REAL;

    IN_Outdoor_Temp : REAL := 0.0;
    IN_Preheat_Request : BOOL := FALSE;
    IN_Freeze_Request : BOOL := FALSE;

    IN_Water_Sensors : ARRAY[1..GVL_CONSTANTS.C_MAX_FLOOD_SENSORS] OF BOOL;
    IN_Smoke_Sensors : ARRAY[1..GVL_CONSTANTS.C_MAX_SMOKE_SENSORS] OF BOOL;
    IN_Methane_Sensors : ARRAY[1..GVL_CONSTANTS.C_MAX_METHANE_SENSORS] OF REAL;
    IN_CO_Sensors : ARRAY[1..GVL_CONSTANTS.C_MAX_CO_SENSORS] OF REAL;

    IN_Input_Degraded : BOOL := FALSE;
    IN_Sensor_Fault : BOOL := FALSE;

    IN_Validation_Failed : BOOL := FALSE;
    IN_Anomaly_Detected : BOOL := FALSE;
    IN_Validation_Reason : STRING(120) := '';
    IN_Anomaly_Reason : STRING(120) := '';
    IN_Last_Invalid_Zone : INT := 0;

    IN_Room_Temp_Prev : ARRAY[1..GVL_CONSTANTS.C_MAX_ZONES] OF REAL;
    IN_Room_Hum_Prev : ARRAY[1..GVL_CONSTANTS.C_MAX_ZONES] OF REAL;
    IN_Last_Change_MS : ARRAY[1..GVL_CONSTANTS.C_MAX_ZONES] OF UDINT;

    IN_Room_Temp_Confidence : ARRAY[1..GVL_CONSTANTS.C_MAX_ZONES] OF REAL;
    IN_Room_Hum_Confidence : ARRAY[1..GVL_CONSTANTS.C_MAX_ZONES] OF REAL;
    IN_Zone_Confidence : ARRAY[1..GVL_CONSTANTS.C_MAX_ZONES] OF REAL;

    // NEW: reputation (long-term learning)
    IN_Room_Temp_Reputation : ARRAY[1..GVL_CONSTANTS.C_MAX_ZONES] OF REAL;
    IN_Room_Hum_Reputation : ARRAY[1..GVL_CONSTANTS.C_MAX_ZONES] OF REAL;

    IN_Min_Zone_Confidence : REAL := 1.0;
    IN_Worst_Zone : INT := 0;
END_VAR

(* ---- GVL_INPUT_VALIDATION_CONFIG.gvl ---- *)
{attribute 'qualified_only'}
VAR_GLOBAL
    // Input validation / temporal anomaly configuration.
    // Used by PRG_Input_Processing only.

    G_Enable_Reputation_Learning : BOOL := TRUE;

    G_Room_Temp_Min : REAL := -40.0;
    G_Room_Temp_Max : REAL := 80.0;
    G_Room_Hum_Min : REAL := 0.0;
    G_Room_Hum_Max : REAL := 100.0;

    G_Room_Temp_Spike_Threshold : REAL := 5.0;
    G_Room_Hum_Spike_Threshold : REAL := 20.0;

    // Confidence/reputation parameters.
    G_Reputation_Learning_Rate : REAL := 0.05;
    G_Reputation_Recovery_Decay : REAL := 0.01;
    G_Min_Sensor_Confidence : REAL := 0.1;
    G_Bad_Spike_Confidence : REAL := 0.3;
    G_Default_Confidence : REAL := 1.0;
END_VAR

(* ---- GVL_INTENT_BEHAVIOR.gvl ---- *)
VAR_GLOBAL
    // Behavior / Scenario Engine intent layer.
    // Scenario Engine writes here; Command Arbitration may consume it.

    I_Request_Night_Mode : BOOL := FALSE;
    I_Request_Away_Mode : BOOL := FALSE;
    I_Request_Comfort_Mode : BOOL := FALSE;
    I_Request_Energy_Save_Mode : BOOL := FALSE;
    I_Request_Preheat : BOOL := FALSE;
    I_Request_Ventilation_Boost : BOOL := FALSE;
    I_Request_Access_Secure_Mode : BOOL := FALSE;

    I_Target_Comfort_Temperature : REAL := 21.0;
    I_Behavior_Priority : INT := 0;

    // Candidate scenario scores for explainability / diagnostics
    I_Score_Comfort : INT := 0;
    I_Score_Night : INT := 0;
    I_Score_Energy_Save : INT := 0;
    I_Score_Preheat : INT := 0;
    I_Score_Vent_Boost : INT := 0;
    I_Score_Access_Secure : INT := 0;

    I_Selected_Scenario_Code : E_System_Reason_Code := REASON_NONE;
    I_Selected_Scenario_Text : STRING(255) := 'No behavior scenario selected';

    I_Reason_Code : E_System_Reason_Code := REASON_NONE;
    I_Reason_Text : STRING(255) := 'No behavior scenario active';
    I_Last_Update_MS : UDINT := 0;
END_VAR

(* ---- GVL_INTENT_SYSTEM.gvl ---- *)
VAR_GLOBAL
    // --- meta ---
    I_Source_Valid : BOOL := FALSE;
    I_Last_Update_Cycle : UDINT := 0;
    I_Last_Update_MS : UDINT := 0;

    // --- system mode constraints ---
    I_Mode_Safe_Stop_Active : BOOL := FALSE;
    I_Mode_Degraded_Active : BOOL := FALSE;
    I_Mode_Freeze_Protection_Active : BOOL := FALSE;

    // --- scenario / automation ---
    I_Preheat_Request : BOOL := FALSE;
    I_Freeze_Request : BOOL := FALSE;
    I_Scenario_Request_Allowed : BOOL := FALSE;

    // --- gateway / system permissions ---
    I_Gateway_Command_Valid : BOOL := FALSE;
    I_Gateway_Command_Type : INT := 0;
    I_Gateway_Writes_Allowed : BOOL := FALSE;
    I_Reset_Errors_Request : BOOL := FALSE;
    I_Config_Apply_Allowed : BOOL := FALSE;
    I_Time_Sync_Allowed : BOOL := FALSE;
    I_Temperature_Write_Allowed : BOOL := FALSE;
    I_Ventilation_Write_Allowed : BOOL := FALSE;
    I_Maintenance_Apply_Allowed : BOOL := FALSE;

    // --- permissions / constraints ---
    I_Access_Open_Allowed : BOOL := FALSE;
    I_Manual_Override_Allowed : BOOL := FALSE;
    I_Dangerous_Action_Allowed : BOOL := FALSE;
END_VAR

(* ---- GVL_INTENT_USER.gvl ---- *)
VAR_GLOBAL
    I_Source_Valid : BOOL := FALSE;
    I_Last_Update_Cycle : UDINT := 0;
    I_Last_Update_MS : UDINT := 0;

    I_Arm_Request : BOOL := FALSE;
    I_Disarm_Request : BOOL := FALSE;

    I_PIN_Code : STRING(8);
    I_RFID_Tag : STRING(32);
    I_2FA_Code_In : STRING(8);

    I_Gate_Open_Request : BOOL := FALSE;
    I_Wicket_Open_Request : BOOL := FALSE;

    I_Lock_1_Open_Request : BOOL := FALSE;
    I_Lock_1_Close_Request : BOOL := FALSE;
    I_Lock_2_Open_Request : BOOL := FALSE;
    I_Lock_2_Close_Request : BOOL := FALSE;

    I_Dangerous_Action_Request : BOOL := FALSE;
    I_Dangerous_Action_Confirm : BOOL := FALSE;
    I_User_Access_Level : INT := 0;

    I_Water_Valve_Test_Open : BOOL := FALSE;
    I_Water_Valve_Test_Close : BOOL := FALSE;
    I_Water_Valve_Test_Confirm : BOOL := FALSE;

    I_Gas_Valve_Test_Open : BOOL := FALSE;
    I_Gas_Valve_Test_Close : BOOL := FALSE;
    I_Gas_Valve_Test_Confirm : BOOL := FALSE;

    I_Water_Selective_Recover : BOOL := FALSE;
    I_Gas_Selective_Recover : BOOL := FALSE;
    I_Scenario_Request : E_SCENARIO_TYPE := E_SCENARIO_TYPE.SCENARIO_NONE;
    I_Lighting_Override_32 : ARRAY[1..GVL_CONSTANTS.C_MAX_LIGHT_ZONES] OF BYTE;
    I_Blinds_Override_32 : ARRAY[1..GVL_CONSTANTS.C_MAX_BLINDS] OF BYTE;
    I_Socket_Override_32 : ARRAY[1..GVL_CONSTANTS.C_MAX_SOCKETS] OF BOOL;
    I_Reset_Errors : BOOL := FALSE;

    I_Set_Temp_Req : BOOL := FALSE;
    I_Target_Zone : INT := 0;
    I_Target_Temperature : REAL := 0.0;
    I_Set_Vent_Req : BOOL := FALSE;
    I_Target_Vent_Speed : REAL := 0.0;
    I_Set_Config_Req : BOOL := FALSE;
    I_Time_Sync_Req : BOOL := FALSE;
    I_New_Time_MS : UDINT := 0;

    I_Set_Adapt_Profile_Req : BOOL := FALSE;
    I_Set_Adapt_Profile_Confirm : BOOL := FALSE;
    I_Adapt_Profile_Value : E_Adapt_Profile := ADAPT_PROFILE_BALANCED;
END_VAR

(* ---- GVL_IO.gvl ---- *)
{attribute 'qualified_only'}
VAR_GLOBAL
    // ======================================================
    // PHYSICAL IO SURFACE
    // ======================================================
    // Input fields are hardware/mapping observations.
    // Output fields are the terminal physical publication surface.
    //
    // PRG_IO_Write is the only runtime-layer publisher for physical
    // output commands in this GVL. Upstream authority/governance,
    // verifier, recovery and observability layers must not write
    // physical outputs directly.
    // ======================================================

    DI_Security_Open : ARRAY[1..GVL_CONSTANTS.C_MAX_SECURITY_SENSORS] OF BOOL;
    DI_Security_Glass : ARRAY[1..GVL_CONSTANTS.C_MAX_SECURITY_SENSORS] OF BOOL;
    DI_Security_2F_Group : BOOL;
    DI_Flood_Sensors : ARRAY[1..GVL_CONSTANTS.C_MAX_FLOOD_SENSORS] OF BOOL;
    DI_Manifold_End_Switches : ARRAY[1..GVL_CONSTANTS.C_MAX_MANIFOLDS] OF BOOL;
    AO_Manifold_Valves : ARRAY[1..GVL_CONSTANTS.C_MAX_MANIFOLDS] OF UINT;
    DO_Manifold_Pumps : ARRAY[1..GVL_CONSTANTS.C_MAX_MANIFOLDS] OF BOOL;
    AI_Manifold_Currents : ARRAY[1..GVL_CONSTANTS.C_MAX_MANIFOLDS] OF INT;
    AI_Manifold_Pressures : ARRAY[1..GVL_CONSTANTS.C_MAX_MANIFOLDS] OF INT;
    AI_Manifold_Temps_Supply : ARRAY[1..GVL_CONSTANTS.C_MAX_MANIFOLDS] OF ST_Owen_Analog_Value;
    AI_Manifold_Temps_Return : ARRAY[1..GVL_CONSTANTS.C_MAX_MANIFOLDS] OF INT;
    AO_Supply_Fans : ARRAY[1..GVL_CONSTANTS.C_MAX_SUPPLY_FANS] OF UINT;
    AO_Exhaust_Fans : ARRAY[1..GVL_CONSTANTS.C_MAX_EXHAUST_FANS] OF UINT;
    AO_Lighting_Levels : ARRAY[1..GVL_CONSTANTS.C_MAX_LIGHT_ZONES] OF UINT;
    AO_Blinds_Positions : ARRAY[1..GVL_CONSTANTS.C_MAX_BLINDS] OF UINT;
    AI_Supply_Temps : ARRAY[1..GVL_CONSTANTS.C_MAX_SUPPLY_TEMPS] OF ST_Owen_Analog_Value;
    AI_Boiler_Modulation : ARRAY[1..GVL_CONSTANTS.C_MAX_BOILERS] OF INT;
    AI_Boiler_Flame_Status : ARRAY[1..GVL_CONSTANTS.C_MAX_BOILERS] OF BOOL;
    DI_Boiler_Error : ARRAY[1..GVL_CONSTANTS.C_MAX_BOILERS] OF BOOL;
    AI_Methane_LEL : ARRAY[1..GVL_CONSTANTS.C_MAX_METHANE_SENSORS] OF ST_Owen_Analog_Value;
    AI_CO_PPM : ARRAY[1..GVL_CONSTANTS.C_MAX_CO_SENSORS] OF REAL;
    DI_Smoke_Sensors : ARRAY[1..GVL_CONSTANTS.C_MAX_SMOKE_SENSORS] OF BOOL;
    AI_Temp_Outdoor : ST_Owen_Analog_Value;
    AI_Floor_Temps : ARRAY[1..GVL_CONSTANTS.C_MAX_ZONES] OF REAL;
    AI_Room_Temps : ARRAY[1..GVL_CONSTANTS.C_MAX_ZONES] OF REAL;
    AI_Room_Hum : ARRAY[1..GVL_CONSTANTS.C_MAX_ZONES] OF REAL;
    AI_Room_CO2 : ARRAY[1..GVL_CONSTANTS.C_MAX_ZONES] OF REAL;
    DO_Zone_Valves : ARRAY[1..GVL_CONSTANTS.C_MAX_HEATING_CIRCUITS] OF BOOL;
    AI_DHW_Temp : REAL;
    AI_DHW_Pressure : REAL;
    DO_DHW_Heating_Pump : BOOL;
    DO_DHW_Circ_Pump : BOOL;
    DO_Backup_Circulation_Pump : BOOL;
    DO_Electric_Heater_Enable : BOOL;
    DI_Lighting_Switches : ARRAY[1..GVL_CONSTANTS.C_MAX_LIGHT_ZONES] OF BOOL;
    DI_Socket_Switches : ARRAY[1..GVL_CONSTANTS.C_MAX_SOCKETS] OF BOOL;
    DI_Motion_Sensors : ARRAY[1..GVL_CONSTANTS.C_MAX_LIGHT_ZONES] OF BOOL;
    DO_Sockets : ARRAY[1..GVL_CONSTANTS.C_MAX_SOCKETS] OF BOOL;
    DO_Gas_Valve_Close : BOOL;

    // Water common inlet valves: 35 = ХВС, 36 = ГВС.
    DO_Water_Valve_35_Open : BOOL;
    DO_Water_Valve_35_Close : BOOL;
    DO_Water_Valve_36_Open : BOOL;
    DO_Water_Valve_36_Close : BOOL;

    // Water local riser valves: 1/2 riser 1, 3/4 riser 2, 5/6 riser 3.
    DO_Water_Local_Valve_Open : ARRAY[1..6] OF BOOL;
    DO_Water_Local_Valve_Close : ARRAY[1..6] OF BOOL;

    AI_Water_Valve_35_Current : REAL;
    AI_Water_Valve_36_Current : REAL;
    DI_Power_OK : BOOL;
    DO_Gas_Siren : BOOL;
    DO_Fire_Siren : BOOL;
    DO_Security_Siren : BOOL;
    DO_Pump_Main_Enable : BOOL;
    DO_Gate_Open : BOOL;
    DO_Wicket_Open : BOOL;
    DO_Lock_1_Open : BOOL;
    DO_Lock_1_Close : BOOL;
    DO_Lock_2_Open : BOOL;
    DO_Lock_2_Close : BOOL;
    DI_Partner_Pulse : BOOL;
    DI_Partner_Active : BOOL;
    DO_Heartbeat_Pulse : BOOL;
    DO_Active_Status : BOOL;
    DI_Module_1_Heartbeat : BOOL;
    DI_Module_2_Heartbeat : BOOL;
    DI_Backup_Circulation_Pump_Feedback : BOOL;
    DI_Electric_Heater_Feedback : BOOL;
    DI_Water_Zone_Open_FB : ARRAY[1..GVL_CONSTANTS.C_MAX_WATER_ZONES] OF BOOL;
    DI_Water_Zone_Close_FB : ARRAY[1..GVL_CONSTANTS.C_MAX_WATER_ZONES] OF BOOL;
    DO_Water_Zone_Enable : ARRAY[1..GVL_CONSTANTS.C_MAX_WATER_ZONES] OF BOOL;
END_VAR

(* ---- GVL_IO_Binding_Config.gvl ---- *)
{attribute 'qualified_only'}
VAR_GLOBAL
    G_Flood_Sensor_Binding : ARRAY[1..64] OF ST_IO_Binding_Record;
    G_Water_Valve_Open_FB_Binding : ARRAY[1..64] OF ST_IO_Binding_Record;
    G_Water_Valve_Close_FB_Binding : ARRAY[1..64] OF ST_IO_Binding_Record;
    G_Water_Valve_Output_Binding : ARRAY[1..64] OF ST_IO_Binding_Record;
END_VAR

VAR_GLOBAL RETAIN
    G_Binding_Config_Version : UDINT;
    G_Binding_Config_Valid : BOOL;
END_VAR

(* ---- GVL_IO_Binding_Runtime.gvl ---- *)
{attribute 'qualified_only'}
VAR_GLOBAL
    G_Runtime_Valid : BOOL;
    G_Last_Update_MS : UDINT;

    G_Any_Invalid_Binding : BOOL;
    G_Any_Missing_Binding : BOOL;

    G_Status_Code : UINT;
    G_Status_Text : STRING(128);
END_VAR

(* ---- GVL_Lifetime.gvl ---- *)
VAR_GLOBAL
    // === LIFETIME STATUS STORAGE ===
    G_Status : ARRAY[1..4] OF ST_Lifetime_Status;

    // === DEVICE IDS ===
    G_Device_Pump : BYTE := 1;
    G_Device_Fan  : BYTE := 2;

    // === HMI / HEALTH READY FLAGS ===
    G_Pump_Maintenance_Required : BOOL;
    G_Fan_Maintenance_Required  : BOOL;

    // === LIFETIME LIMITS ===
    G_Pump_Nominal_Hours : UDINT := 10000;
    G_Fan_Nominal_Hours  : UDINT := 15000;

    // === WARNING THRESHOLDS ===
    G_Maintenance_Threshold_Percent : BYTE := 20;

    // === HMI ACTIVE VIEW ===
    G_Active_Device_Index : INT := 1;
    G_Active_Runtime_Hours : UDINT;
    G_Active_Remaining_Hours : UDINT;
    G_Active_Remaining_Percent : BYTE;
    G_Active_Maintenance_Required : BOOL;

    // === HMI LABELS ===
    G_Device1_Label : STRING(32) := 'Pump';
    G_Device2_Label : STRING(32) := 'Vent Fan';
    G_Active_Label : STRING(32);

    // === RESERVED DEVICE IDS ===
    G_Device_Reserved_3 : BYTE := 3;
    G_Device_Reserved_4 : BYTE := 4;

    // === HMI LABEL ARRAY ===
    G_Device_Labels : ARRAY[1..4] OF STRING(32) := ['Pump', 'Vent Fan', 'Reserved 3', 'Reserved 4'];

    // === HEALTH SUMMARY ===
    G_Any_Maintenance_Required : BOOL;
    G_Maintenance_Warning : BOOL;
    G_Maintenance_Critical : BOOL;

END_VAR

(* ---- GVL_MAIN_PHASE_FEEDBACK.gvl ---- *)
{attribute 'qualified_only'}
VAR_GLOBAL
    // MAIN phase feedback is observational only.
    // It does not gate execution and does not control physical outputs.

    G_Cycle_Start_MS : UDINT;
    G_Last_Update_MS : UDINT;
    G_Current_Phase : UINT;

    G_Phase_01_Bootstrap_Executed : BOOL;
    G_Phase_01_Bootstrap_Valid : BOOL;
    G_Phase_01_Bootstrap_Status_Text : STRING(128);

    G_Phase_02_Redundancy_Executed : BOOL;
    G_Phase_02_Redundancy_Valid : BOOL;
    G_Phase_02_Redundancy_Status_Text : STRING(128);

    G_Phase_03_Input_Safety_Command_Executed : BOOL;
    G_Phase_03_Input_Safety_Command_Valid : BOOL;
    G_Phase_03_Input_Safety_Command_Status_Text : STRING(128);

    G_Phase_04_Transport_Distributed_Executed : BOOL;
    G_Phase_04_Transport_Distributed_Valid : BOOL;
    G_Phase_04_Transport_Distributed_Status_Text : STRING(128);

    G_Phase_05_Domain_Output_Executed : BOOL;
    G_Phase_05_Domain_Output_Valid : BOOL;
    G_Phase_05_Domain_Output_Status_Text : STRING(128);

    G_Phase_06_PostOutput_Authority_Executed : BOOL;
    G_Phase_06_PostOutput_Authority_Valid : BOOL;
    G_Phase_06_PostOutput_Authority_Status_Text : STRING(128);

    G_Phase_07_Semantic_Governance_Executed : BOOL;
    G_Phase_07_Semantic_Governance_Valid : BOOL;
    G_Phase_07_Semantic_Governance_Status_Text : STRING(128);

    G_Phase_07_Full_Semantic_Requested : BOOL;
    G_Phase_07_Full_Semantic_Executed : BOOL;
    G_Phase_07_Full_Semantic_Skipped_By_Design : BOOL;

    G_Phase_07_Extended_Observability_Requested : BOOL;
    G_Phase_07_Extended_Observability_Executed : BOOL;
    G_Phase_07_Extended_Observability_Skipped_By_Design : BOOL;

    G_Phase_07_Analytics_Requested : BOOL;
    G_Phase_07_Analytics_Executed : BOOL;
    G_Phase_07_Analytics_Skipped_By_Design : BOOL;

    G_Phase_08_Diagnostics_HMI_Executed : BOOL;
    G_Phase_08_Diagnostics_HMI_Valid : BOOL;
    G_Phase_08_Diagnostics_HMI_Status_Text : STRING(128);

    G_Phase_08_Extended_Diagnostics_Requested : BOOL;
    G_Phase_08_Extended_Diagnostics_Executed : BOOL;
    G_Phase_08_Extended_Diagnostics_Skipped_By_Design : BOOL;

    G_Phase_08_Extended_Observability_Requested : BOOL;
    G_Phase_08_Extended_Observability_Executed : BOOL;
    G_Phase_08_Extended_Observability_Skipped_By_Design : BOOL;

    G_Phase_08_Simulation_Requested : BOOL;
    G_Phase_08_Simulation_Executed : BOOL;
    G_Phase_08_Simulation_Skipped_By_Design : BOOL;

    G_Critical_Path_Executed : BOOL;
    G_Critical_Path_Valid : BOOL;
    G_Observability_Path_Executed : BOOL;
    G_Observability_Path_Valid : BOOL;
    G_Any_Phase_Invalid : BOOL;
    G_Any_Phase_Skipped_By_Design : BOOL;
    G_Status_Code : UINT;
    G_Status_Text : STRING(160);
END_VAR

(* ---- GVL_METHANE_REDUNDANCY.gvl ---- *)
{attribute 'qualified_only'}
VAR_GLOBAL
    G_Sensor_1_LEL : REAL := 0.0;
    G_Sensor_2_LEL : REAL := 0.0;
    G_Max_LEL : REAL := 0.0;
    G_Min_LEL : REAL := 0.0;
    G_Diff_LEL : REAL := 0.0;
    G_Max_Sensor_Index : INT := 0;
    G_Disagreement_Active : BOOL := FALSE;
    G_Disagreement_Limit_LEL : REAL := 5.0;
    G_Redundancy_Available : BOOL := FALSE;
    G_Conservative_Max_Selected : BOOL := TRUE;
    G_Status_Text : STRING(160) := 'Methane redundancy idle';
    G_Last_Update_MS : UDINT := 0;
END_VAR

(* ---- GVL_MODBUS_MASTER.gvl ---- *)
{attribute 'qualified_only'}
VAR_GLOBAL
    // ======================================================
    // MODBUS MASTER RUNTIME CONTRACT
    // ======================================================
    // This layer is intentionally library-independent.
    // Concrete CODESYS Modbus RTU implementation consumes Request[]
    // via GVL_MODBUS_RTU_BRIDGE and publishes confirmed Response[].

    G_Request : ARRAY[1..16] OF ST_Modbus_Request;
    G_Response : ARRAY[1..16] OF ST_Modbus_Response;

    G_Master_Online : BOOL := FALSE;
    G_Master_Error : BOOL := FALSE;
    G_Last_Transaction_MS : UDINT := 0;

    // Active transaction scheduler state
    G_Active : BOOL := FALSE;
    G_Active_Index : INT := 0;
    G_Active_Sequence : UDINT := 0;
    G_Active_Start_MS : UDINT := 0;
    G_Active_Retry_Count : INT := 0;
    G_Total_Transactions : UDINT := 0;
    G_Total_Errors : UDINT := 0;
    G_Total_Timeouts : UDINT := 0;
END_VAR

(* ---- GVL_MODBUS_RTU_BRIDGE.gvl ---- *)
{attribute 'qualified_only'}
VAR_GLOBAL
    // ======================================================
    // MODBUS RTU BRIDGE CONTRACT
    // ======================================================
    // This GVL is the boundary between project logic and a concrete
    // CODESYS/vendor Modbus Serial Master implementation.
    //
    // Project side writes Request_*.
    // Concrete RTU driver writes Response_*.
    // No fake Done is produced here.

    G_Bridge_Enabled : BOOL := FALSE;
    G_Driver_Online : BOOL := FALSE;
    G_Driver_Error : BOOL := FALSE;
    G_Driver_Error_Code : WORD := 0;

    G_Request_Valid : BOOL := FALSE;
    G_Request_Index : INT := 0;
    G_Request_Slave_ID : BYTE := 0;
    G_Request_Function_Code : E_Modbus_Function := MB_NONE;
    G_Request_Start_Register : UINT := 0;
    G_Request_Register_Count : UINT := 0;
    G_Request_Write_Value : ARRAY[1..32] OF WORD;
    G_Request_Sequence : UDINT := 0;
    G_Request_Timeout_MS : UDINT := 0;

    G_Response_Busy : BOOL := FALSE;
    G_Response_Done : BOOL := FALSE;
    G_Response_Error : BOOL := FALSE;
    G_Response_Error_Code : WORD := 0;
    G_Response_Value : ARRAY[1..32] OF WORD;
    G_Response_Sequence : UDINT := 0;
    G_Response_Update_MS : UDINT := 0;
END_VAR

(* ---- GVL_MODBUS_SYSCOM_TRANSPORT.gvl ---- *)
{attribute 'qualified_only'}
VAR_GLOBAL
    // ======================================================
    // MODBUS RTU SYSCOM BYTE TRANSPORT BOUNDARY
    // ======================================================

    G_Transport_Attached : BOOL := FALSE;

    // Backend runtime/reconnect state
    G_Backend_State : E_Modbus_SysCom_Backend_State := MB_SYSCOM_CLOSED;
    G_Backend_Last_Error_MS : UDINT := 0;
    G_Backend_Reconnect_Delay_MS : UDINT := 3000;
    G_Backend_Reconnect_Attempts : UDINT := 0;
    G_Backend_Online : BOOL := FALSE;

    // TX runtime
    G_TX_Request : BOOL := FALSE;
    G_TX_Buffer : ARRAY[0..255] OF BYTE;
    G_TX_Length : UINT := 0;
    G_TX_Done : BOOL := FALSE;
    G_TX_Error : BOOL := FALSE;
    G_TX_Error_Code : WORD := 0;

    // RX runtime
    G_RX_Ready : BOOL := FALSE;
    G_RX_Buffer : ARRAY[0..255] OF BYTE;
    G_RX_Length : UINT := 0;
    G_RX_Error : BOOL := FALSE;

    // RX assembler/runtime state
    G_RX_State : E_Modbus_RTU_RX_State := MB_RTU_RX_IDLE;

    G_RX_Assembler_Active : BOOL := FALSE;
    G_RX_Assembler_Length : UINT := 0;
    G_RX_Assembler_Last_Byte_MS : UDINT := 0;
    G_RX_Assembler_InterFrame_MS : UDINT := 20;
    G_RX_Assembler_Overflow : BOOL := FALSE;
    G_RX_Assembler_CRC_OK : BOOL := FALSE;
    G_RX_Assembler_CRC_Frame : WORD := 0;
    G_RX_Assembler_CRC_Calc : WORD := 0;

    // Watchdog timestamps
    G_Last_TX_Request_MS : UDINT := 0;
    G_Last_TX_Done_MS : UDINT := 0;
    G_Last_RX_MS : UDINT := 0;

    // Runtime watchdog flags
    G_TX_Watchdog_Timeout : BOOL := FALSE;
    G_RX_Watchdog_Timeout : BOOL := FALSE;
    G_Bus_Silent : BOOL := FALSE;

    // Statistics
    G_Total_TX : UDINT := 0;
    G_Total_RX : UDINT := 0;
    G_Total_Errors : UDINT := 0;
    G_Total_RX_Overflow : UDINT := 0;
    G_Total_RX_Short_Frame : UDINT := 0;
    G_Total_RX_CRC_Error : UDINT := 0;
    G_Total_Reconnects : UDINT := 0;
    G_Total_TX_Watchdog : UDINT := 0;
    G_Total_RX_Watchdog : UDINT := 0;
END_VAR

(* ---- GVL_MODE.gvl ---- *)
{attribute 'qualified_only'}
VAR_GLOBAL
    G_Current_Behavior_Mode : E_Behavior_Mode := BEHAVIOR_HOME;
    G_Mode_Last_Change_TS : UDINT := 0;
    G_Mode_Code : UDINT := 0;
END_VAR

(* ---- GVL_OBSERVABILITY_AUTHORITY.gvl ---- *)
VAR_GLOBAL
    // ======================================================
    // OBSERVABILITY VISIBILITY STATE
    // ======================================================

    Observability_Epoch : ULINT := 0;
    Observability_Snapshot_Epoch : ULINT := 0;

    Publication_Runtime_Valid : BOOL := FALSE;

    Unsafe_State_Published : BOOL := FALSE;
    Emergency_Visibility_Required : BOOL := FALSE;

    Runtime_Failure_Visible : BOOL := FALSE;
    Output_Decay_Visible : BOOL := FALSE;
    Transport_Failure_Visible : BOOL := FALSE;
    Recovery_Failure_Visible : BOOL := FALSE;
    Fencing_Failure_Visible : BOOL := FALSE;
    Monotonic_Failure_Visible : BOOL := FALSE;

    Distributed_Failure_Visible : BOOL := FALSE;
    Distributed_Quarantine_Visible : BOOL := FALSE;
    Peer_Runtime_Stale_Visible : BOOL := FALSE;
    Peer_Snapshot_Stale_Visible : BOOL := FALSE;
    Peer_Boot_Mismatch_Visible : BOOL := FALSE;
    Peer_Fencing_Conflict_Visible : BOOL := FALSE;
    Peer_Semantic_Continuity_Lost_Visible : BOOL := FALSE;

    Distributed_Publication_Reconciliation_Visible : BOOL := FALSE;
    Distributed_Publication_Freeze_Visible : BOOL := FALSE;
    Distributed_Snapshot_Consistency_Visible : BOOL := FALSE;

    Peer_Publication_Stale_Visible : BOOL := FALSE;
    Peer_Publication_Divergence_Visible : BOOL := FALSE;
    Peer_Publication_Reconciliation_Lost_Visible : BOOL := FALSE;
    Peer_Snapshot_Not_Immutable_Visible : BOOL := FALSE;

    Distributed_Immutable_Snapshot_Quarantine_Visible : BOOL := FALSE;

    Distributed_Commit_Visible : BOOL := FALSE;
    Distributed_Commit_Quarantine_Visible : BOOL := FALSE;

    Publication_Prepare_Visible : BOOL := FALSE;
    Publication_Commit_Visible : BOOL := FALSE;

    Peer_Commit_Ack_Visible : BOOL := FALSE;
    Peer_Commit_Mismatch_Visible : BOOL := FALSE;
    Peer_Commit_Replay_Visible : BOOL := FALSE;
    Peer_Commit_Missing_Visible : BOOL := FALSE;

    Commit_Lease_Expired_Visible : BOOL := FALSE;

    Observability_Last_Publication_MS : UDINT := 0;

    Observability_Last_Error_Code : UDINT := 0;
    Observability_Last_Error_Text : STRING(160) := '';
END_VAR

(* ---- GVL_OBSERVABILITY_AUTHORITY_FABRIC.gvl ---- *)
VAR_GLOBAL
    // Global observability authority.
    Observability_Authority_Valid : BOOL := FALSE;
    Observability_Quarantine_Active : BOOL := TRUE;
    Observability_Publication_Allowed : BOOL := FALSE;

    // Authority-aware observability.
    HMI_Authority_Coherent : BOOL := FALSE;
    Diagnostics_Authority_Coherent : BOOL := FALSE;
    Blackbox_Authority_Coherent : BOOL := FALSE;
    Trend_Authority_Coherent : BOOL := FALSE;
    Alarm_Authority_Coherent : BOOL := FALSE;

    // Stale observability detection.
    Stale_HMI_State_Detected : BOOL := FALSE;
    Diagnostic_Epoch_Skew_Detected : BOOL := FALSE;
    Post_Revocation_Observability_Lag : BOOL := FALSE;
    Nonauthoritative_Operator_State_Detected : BOOL := FALSE;

    // Epoch coherence.
    Observability_Epoch : UDINT := 0;
    Observability_Epoch_Coherent : BOOL := FALSE;

    // Temporal authority.
    Observability_Last_Update_MS : UDINT := 0;
    Observability_Lease_Expired : BOOL := TRUE;

    // Diagnostics.
    Observability_Last_Error_Code : UDINT := 0;
    Observability_Last_Error_Text : STRING(160) := '';
    Observability_Invalidation_Count : UDINT := 0;
END_VAR

(* ---- GVL_OPENTHERM_ADAPTER.gvl ---- *)
{attribute 'qualified_only'}
VAR_GLOBAL
    // ======================================================
    // PHYSICAL OPENTHERM ADAPTER CONTRACT
    // ======================================================
    // Commands are written by FB_Boiler_OpenTherm_Interface.
    // Raw status fields are updated by PRG_OpenTherm_Transport.

    G_Command : ARRAY[1..GVL_CONSTANTS.C_MAX_BOILERS] OF ST_OpenTherm_Command;
    G_Status : ARRAY[1..GVL_CONSTANTS.C_MAX_BOILERS] OF ST_OpenTherm_Status;

    // Transport layer register mapping
    G_Register_Map : ARRAY[1..GVL_CONSTANTS.C_MAX_BOILERS] OF ST_OpenTherm_Register_Map;

    // Raw wire image exchanged with transport layer
    G_Wire_Image : ARRAY[1..GVL_CONSTANTS.C_MAX_BOILERS] OF ST_OpenTherm_Wire_Image;

    // Transport diagnostics
    G_Transport_Online : BOOL := FALSE;
    G_Transport_Error : BOOL := FALSE;
    G_Last_Transport_Update_MS : UDINT := 0;

    // Timing configuration
    G_Heartbeat_Timeout_MS : UDINT := 5000;
    G_Command_Ack_Timeout_MS : UDINT := 3000;
END_VAR

(* ---- GVL_OUTPUT_EPOCH.gvl ---- *)
VAR_GLOBAL
    // ======================================================
    // OUTPUT PUBLICATION AUTHORITY STATE
    // ======================================================
    // Centralized final physical publication arbitration state.
    //
    // Output_Forced_Safe_Decay is the final output hard-stop
    // authority exported to IO_Write.
    //
    // Output_Publication_Valid / lease / stale fields are
    // derived publication diagnostics and observability state.
    // They must not be reinterpreted by IO_Write as separate
    // hard-stop authorities.
    // ======================================================

    Output_Publication_Epoch : ULINT := 0;
    Output_Publication_Valid : BOOL := FALSE;

    Output_Lease_Active : BOOL := FALSE;
    Output_Lease_Expired : BOOL := FALSE;
    Output_Lease_Timeout_MS : UDINT := 3000;

    Output_Last_Publication_MS : UDINT := 0;
    Output_Last_Refresh_MS : UDINT := 0;
    Output_Last_Invalidation_MS : UDINT := 0;

    Output_Runtime_Epoch : ULINT := 0;
    Output_Runtime_Epoch_Valid : BOOL := FALSE;

    Output_Stale_Detected : BOOL := FALSE;
    Output_Forced_Safe_Decay : BOOL := FALSE;

    // Advisory-only semantic continuity visibility.
    // Does not hard-stop physical output publication.
    Output_Semantic_Continuity_Warning : BOOL := FALSE;

    Output_Last_Error_Code : UDINT := 0;
    Output_Last_Error_Text : STRING(160) := '';
END_VAR

(* ---- GVL_PEER_SESSION.gvl ---- *)
VAR_GLOBAL
    // ======================================================
    // PEER SESSION TRANSPORT CONTRACT
    // ======================================================
    // Transport-neutral remote PLC session exchange surface.
    //
    // Purpose:
    // provide explicit remote runtime/session state for
    // distributed peer ingestion and reconciliation.
    //
    // Ownership:
    // - transport/replication layer publishes Remote_* fields
    // - PRG_Distributed_Peer_Ingestion consumes them
    // - distributed governors must not publish transport state
    //
    // Current state:
    // foundation contract only.
    // explicit network/session replication transport is not yet
    // implemented.
    // ======================================================

    Remote_Session_Valid : BOOL := FALSE;
    Remote_Last_Refresh_MS : UDINT := 0;

    Remote_Runtime_Epoch : ULINT := 0;
    Remote_Snapshot_Epoch : ULINT := 0;
    Remote_Boot_Generation : ULINT := 0;
    Remote_Fencing_Token : ULINT := 0;

    Remote_Publication_Allowed : BOOL := FALSE;
    Remote_Runtime_Healthy : BOOL := FALSE;
END_VAR

(* ---- GVL_PHYSICAL_DEADLOCK_RESOLUTION_FABRIC.gvl ---- *)
VAR_GLOBAL
    Physical_Deadlock_Resolution_Valid : BOOL := FALSE;
    Physical_Deadlock_Resolution_Granted : BOOL := FALSE;

    Deadlock_Resolution_Canonical : BOOL := FALSE;
    Physical_Forward_Progress_Valid : BOOL := FALSE;
    CrossDomain_Execution_Progress_Stable : BOOL := FALSE;
    Recovery_Progress_Stable : BOOL := FALSE;

    Deadlock_Causality_Grounded : BOOL := FALSE;
    Distributed_Deadlock_Consensus_Valid : BOOL := FALSE;

    Physical_CircularWait_Detected : BOOL := FALSE;
    CrossDomain_Progress_Deadlock : BOOL := FALSE;
    Recovery_Livelock_Detected : BOOL := FALSE;
    Physical_Progress_Stall_Detected : BOOL := FALSE;

    Physical_Deadlock_Resolution_Epoch : UDINT := 0;
END_VAR

(* ---- GVL_PHYSICAL_REALITY_VERIFICATION_FABRIC.gvl ---- *)
VAR_GLOBAL
    Physical_Reality_Verification_Active : BOOL := TRUE;
    Physical_Reality_Verification_ReadOnly : BOOL := TRUE;
    Physical_Reality_Verification_NoMutation : BOOL := TRUE;

    Commanded_State_Verified_Physically : BOOL := FALSE;
    Physical_Response_Coherent : BOOL := FALSE;
    Sensor_Physics_Coherent : BOOL := FALSE;
    Physical_Runtime_Reality_Valid : BOOL := FALSE;

    Physical_Reality_Divergence_Detected : BOOL := FALSE;
    Commanded_State_Mismatch_Detected : BOOL := FALSE;
    Impossible_Physical_Response_Detected : BOOL := FALSE;
    Sensor_Physics_Contradiction_Detected : BOOL := FALSE;

    Passive_Physics_Reasoning_Active : BOOL := TRUE;
    Physical_Contradiction_Observed : BOOL := FALSE;

    Physical_Reality_Verification_Epoch : UDINT := 0;
END_VAR
